LIN {X 0,Y 384.347,Z 411.583,A -85,B 0,C 180,E1 -11892.675,E2 -11892.675} C_VEL
LIN {X 0,Y 385.318,Z 404.439,A -85,B 0,C 180,E1 -11894.524,E2 -11894.524} C_VEL
LIN {X 0,Y 386.67,Z 395.805,A -85,B 0,C 180,E1 -11896.363,E2 -11896.363} C_VEL
LIN {X 0,Y 388.197,Z 385.439,A -85,B 0,C 180,E1 -11898.197,E2 -11898.197} C_VEL
LIN {X 0,Y 389.705,Z 374.807,A -85,B 0,C 180,E1 -11899.763,E2 -11899.763} C_VEL
LIN {X 0,Y 391.478,Z 362.137,A -85,B 0,C 180,E1 -11901.317,E2 -11901.317} C_VEL
LIN {X 0,Y 393.105,Z 349.489,A -85,B 0,C 180,E1 -11902.605,E2 -11902.605} C_VEL
LIN {X 0,Y 394.718,Z 335.76,A -85,B 0,C 180,E1 -11903.756,E2 -11903.756} C_VEL
LIN {X 0,Y 396.173,Z 321.35,A -85,B 0,C 180,E1 -11904.735,E2 -11904.735} C_VEL
LIN {X 0,Y 397.574,Z 305.833,A -85,B 0,C 180,E1 -11905.551,E2 -11905.551} C_VEL
LIN {X 0,Y 398.601,Z 290.565,A -85,B 0,C 180,E1 -11906.154,E2 -11906.154} C_VEL
LIN {X 0,Y 403.483,Z 217.535,A -85,B 0,C 180,E1 -11908.256,E2 -11908.256} C_VEL
LIN {X 0,Y 407.824,Z 166.369,A -85,B 0,C 180,E1 -11909.77,E2 -11909.77} C_VEL
LIN {X 0,Y 404.879,Z 160.3,A -85,B 0,C 180,E1 -11910.501,E2 -11910.501} C_VEL
LIN {X 0,Y 400.279,Z 152.554,A -85,B 0,C 180,E1 -11911.666,E2 -11911.666} C_VEL
LIN {X 0,Y 396.216,Z 146.476,A -85,B 0,C 180,E1 -11912.795,E2 -11912.795} C_VEL
LIN {X 0,Y 393.462,Z 142.689,A -85,B 0,C 180,E1 -11913.622,E2 -11913.622} C_VEL
LIN {X 0,Y 390.258,Z 138.514,A -85,B 0,C 180,E1 -11914.697,E2 -11914.697} C_VEL
LIN {X 0,Y 387.178,Z 134.685,A -85,B 0,C 180,E1 -11915.863,E2 -11915.863} C_VEL
LIN {X 0,Y 386.326,Z 132.28,A -85,B 0,C 180,E1 -11918.208,E2 -11918.208} C_VEL
LIN {X 0,Y 385.813,Z 130.877,A -85,B 0,C 180,E1 -11920.978,E2 -11920.978} C_VEL
LIN {X 0,Y 385.849,Z 130.902,A -85,B 0,C 180,E1 -11923.233,E2 -11923.233} C_VEL
LIN {X 0,Y 386.163,Z 131.856,A -85,B 0,C 180,E1 -11925.217,E2 -11925.217} C_VEL
LIN {X 0,Y 386.644,Z 133,A -85,B 0,C 180,E1 -11926.642,E2 -11926.642} C_VEL
LIN {X 0,Y 388.078,Z 136.761,A -85,B 0,C 180,E1 -11929.518,E2 -11929.518} C_VEL
LIN {X 0,Y 389.912,Z 141.995,A -85,B 0,C 180,E1 -11932.205,E2 -11932.205} C_VEL
LIN {X 0,Y 392.082,Z 149.259,A -85,B 0,C 180,E1 -11934.999,E2 -11934.999} C_VEL
LIN {X 0,Y 392.656,Z 151.099,A -85,B 0,C 180,E1 -11935.562,E2 -11935.562} C_VEL
LIN {X 0,Y 396.501,Z 158.649,A -85,B 0,C 180,E1 -11936.812,E2 -11936.812} C_VEL
LIN {X 0,Y 399.421,Z 164.695,A -85,B 0,C 180,E1 -11937.673,E2 -11937.673} C_VEL
LIN {X 0,Y 401.08,Z 168.627,A -85,B 0,C 180,E1 -11938.149,E2 -11938.149} C_VEL
LIN {X 0,Y 403.406,Z 182.486,A -85,B 0,C 180,E1 -11939.166,E2 -11939.166} C_VEL
LIN {X 0,Y 405.189,Z 197.13,A -85,B 0,C 180,E1 -11940.051,E2 -11940.051} C_VEL
LIN {X 0,Y 405.664,Z 204.273,A -85,B 0,C 180,E1 -11940.413,E2 -11940.413} C_VEL
LIN {X 0,Y 399.813,Z 285.015,A -85,B 0,C 180,E1 -11942.733,E2 -11942.733} C_VEL
LIN {X 0,Y 397.323,Z 326,A -85,B 0,C 180,E1 -11943.896,E2 -11943.896} C_VEL
LIN {X 0,Y 395.753,Z 342.836,A -85,B 0,C 180,E1 -11944.562,E2 -11944.562} C_VEL
LIN {X 0,Y 394.082,Z 357.859,A -85,B 0,C 180,E1 -11945.355,E2 -11945.355} C_VEL
LIN {X 0,Y 392.334,Z 372.724,A -85,B 0,C 180,E1 -11946.353,E2 -11946.353} C_VEL
LIN {X 0,Y 389.831,Z 393.298,A -85,B 0,C 180,E1 -11948.032,E2 -11948.032} C_VEL
LIN {X 0,Y 388.472,Z 405.12,A -85,B 0,C 180,E1 -11949.204,E2 -11949.204} C_VEL
LIN {X 0,Y 387.036,Z 417.181,A -85,B 0,C 180,E1 -11950.647,E2 -11950.647} C_VEL
LIN {X 0,Y 385.642,Z 428.175,A -85,B 0,C 180,E1 -11952.226,E2 -11952.226} C_VEL
LIN {X 0,Y 384.521,Z 437.485,A -85,B 0,C 180,E1 -11953.816,E2 -11953.816} C_VEL
LIN {X 0,Y 383.443,Z 446.573,A -85,B 0,C 180,E1 -11955.674,E2 -11955.674} C_VEL
LIN {X 0,Y 382.616,Z 455.061,A -85,B 0,C 180,E1 -11957.805,E2 -11957.805} C_VEL
LIN {X 0,Y 382.021,Z 461.857,A -85,B 0,C 180,E1 -11959.935,E2 -11959.935} C_VEL
LIN {X 0,Y 381.784,Z 467.162,A -85,B 0,C 180,E1 -11962.064,E2 -11962.064} C_VEL
LIN {X 0,Y 381.668,Z 470.632,A -85,B 0,C 180,E1 -11963.906,E2 -11963.906} C_VEL
LIN {X 0,Y 381.614,Z 473.177,A -85,B 0,C 180,E1 -11965.775,E2 -11965.775} C_VEL
LIN {X 0,Y 381.625,Z 474.929,A -85,B 0,C 180,E1 -11967.889,E2 -11967.889} C_VEL
LIN {X 0,Y 381.641,Z 475.494,A -85,B 0,C 180,E1 -11970,E2 -11970} C_VEL
LIN {X 0,Y 381.625,Z 474.855,A -85,B 0,C 180,E1 -11972.111,E2 -11972.111} C_VEL
LIN {X 0,Y 381.618,Z 472.984,A -85,B 0,C 180,E1 -11974.225,E2 -11974.225} C_VEL
LIN {X 0,Y 381.704,Z 469.874,A -85,B 0,C 180,E1 -11976.343,E2 -11976.343} C_VEL
LIN {X 0,Y 381.791,Z 465.448,A -85,B 0,C 180,E1 -11978.468,E2 -11978.468} C_VEL
LIN {X 0,Y 382.103,Z 459.605,A -85,B 0,C 180,E1 -11980.599,E2 -11980.599} C_VEL
LIN {X 0,Y 382.631,Z 453.192,A -85,B 0,C 180,E1 -11982.464,E2 -11982.464} C_VEL
LIN {X 0,Y 383.329,Z 445.398,A -85,B 0,C 180,E1 -11984.33,E2 -11984.33} C_VEL
LIN {X 0,Y 384.374,Z 435.976,A -85,B 0,C 180,E1 -11986.191,E2 -11986.191} C_VEL
LIN {X 0,Y 385.486,Z 426.338,A -85,B 0,C 180,E1 -11987.781,E2 -11987.781} C_VEL
LIN {X 0,Y 386.647,Z 415.895,A -85,B 0,C 180,E1 -11989.236,E2 -11989.236} C_VEL
LIN {X 0,Y 387.865,Z 404.637,A -85,B 0,C 180,E1 -11990.553,E2 -11990.553} C_VEL
LIN {X 0,Y 389.212,Z 392.493,A -85,B 0,C 180,E1 -11991.726,E2 -11991.726} C_VEL
LIN {X 0,Y 391.575,Z 372.289,A -85,B 0,C 180,E1 -11993.398,E2 -11993.398} C_VEL
LIN {X 0,Y 393.335,Z 357.326,A -85,B 0,C 180,E1 -11994.406,E2 -11994.406} C_VEL
LIN {X 0,Y 394.983,Z 341.955,A -85,B 0,C 180,E1 -11995.209,E2 -11995.209} C_VEL
LIN {X 0,Y 396.443,Z 325.504,A -85,B 0,C 180,E1 -11995.848,E2 -11995.848} C_VEL
LIN {X 0,Y 402.25,Z 235.432,A -85,B 0,C 180,E1 -11998.413,E2 -11998.413} C_VEL
LIN {X 0,Y 405.001,Z 198.369,A -85,B 0,C 180,E1 -11999.525,E2 -11999.525} C_VEL
LIN {X 0,Y 403.865,Z 178.688,A -85,B 0,C 180,E1 -12000.517,E2 -12000.517} C_VEL
LIN {X 0,Y 402.692,Z 165.49,A -85,B 0,C 180,E1 -12001.295,E2 -12001.295} C_VEL
LIN {X 0,Y 399.155,Z 154.868,A -85,B 0,C 180,E1 -12002.419,E2 -12002.419} C_VEL
LIN {X 0,Y 395.258,Z 143.156,A -85,B 0,C 180,E1 -12003.828,E2 -12003.828} C_VEL
LIN {X 0,Y 393.762,Z 140.224,A -85,B 0,C 180,E1 -12004.414,E2 -12004.414} C_VEL
LIN {X 0,Y 392.349,Z 137.801,A -85,B 0,C 180,E1 -12004.974,E2 -12004.974} C_VEL
LIN {X 0,Y 391.308,Z 136.6,A -85,B 0,C 180,E1 -12005.364,E2 -12005.364} C_VEL
LIN {X 0,Y 389.233,Z 133.196,A -85,B 0,C 180,E1 -12006.312,E2 -12006.312} C_VEL
LIN {X 0,Y 387.579,Z 131.177,A -85,B 0,C 180,E1 -12007.075,E2 -12007.075} C_VEL
LIN {X 0,Y 386.337,Z 128.589,A -85,B 0,C 180,E1 -12007.852,E2 -12007.852} C_VEL
LIN {X 0,Y 384.354,Z 126.735,A -85,B 0,C 180,E1 -12008.944,E2 -12008.944} C_VEL
LIN {X 0,Y 383.217,Z 124.543,A -85,B 0,C 180,E1 -12009.932,E2 -12009.932} C_VEL
LIN {X 0,Y 382.968,Z 123.404,A -85,B 0,C 180,E1 -12010.424,E2 -12010.424} C_VEL
LIN {X 0,Y 383.005,Z 123.401,A -85,B 0,C 180,E1 -12012.779,E2 -12012.779} C_VEL
LIN {X 0,Y 382.989,Z 123.398,A -85,B 0,C 180,E1 -12015.788,E2 -12015.788} C_VEL
LIN {X 0,Y 382.96,Z 123.404,A -85,B 0,C 180,E1 -12018.801,E2 -12018.801} C_VEL
LIN {X 0,Y 383.017,Z 123.514,A -85,B 0,C 180,E1 -12020.792,E2 -12020.792} C_VEL
LIN {X 0,Y 383.818,Z 125.952,A -85,B 0,C 180,E1 -12021.94,E2 -12021.94} C_VEL
LIN {X 0,Y 385.61,Z 128.057,A -85,B 0,C 180,E1 -12023.315,E2 -12023.315} C_VEL
LIN {X 0,Y 386.401,Z 130.05,A -85,B 0,C 180,E1 -12023.996,E2 -12023.996} C_VEL
LIN {X 0,Y 389.987,Z 134.512,A -85,B 0,C 180,E1 -12025.361,E2 -12025.361} C_VEL
LIN {X 0,Y 393.017,Z 138.694,A -85,B 0,C 180,E1 -12026.39,E2 -12026.39} C_VEL
LIN {X 0,Y 396.646,Z 144.079,A -85,B 0,C 180,E1 -12027.49,E2 -12027.49} C_VEL
LIN {X 0,Y 401.33,Z 151.497,A -85,B 0,C 180,E1 -12028.756,E2 -12028.756} C_VEL
LIN {X 0,Y 406.014,Z 160.362,A -85,B 0,C 180,E1 -12029.938,E2 -12029.938} C_VEL
LIN {X 0,Y 407.556,Z 163.653,A -85,B 0,C 180,E1 -12030.318,E2 -12030.318} C_VEL
LIN {X 0,Y 401.249,Z 243.859,A -85,B 0,C 180,E1 -12032.663,E2 -12032.663} C_VEL
LIN {X 0,Y 398.178,Z 293.464,A -85,B 0,C 180,E1 -12034.088,E2 -12034.088} C_VEL
LIN {X 0,Y 397.002,Z 309.399,A -85,B 0,C 180,E1 -12034.762,E2 -12034.762} C_VEL
LIN {X 0,Y 395.647,Z 324.606,A -85,B 0,C 180,E1 -12035.623,E2 -12035.623} C_VEL
LIN {X 0,Y 394.22,Z 338.624,A -85,B 0,C 180,E1 -12036.63,E2 -12036.63} C_VEL
LIN {X 0,Y 392.635,Z 351.845,A -85,B 0,C 180,E1 -12037.782,E2 -12037.782} C_VEL
LIN {X 0,Y 390.896,Z 365.316,A -85,B 0,C 180,E1 -12039.215,E2 -12039.215} C_VEL
LIN {X 0,Y 389.398,Z 375.479,A -85,B 0,C 180,E1 -12040.495,E2 -12040.495} C_VEL
LIN {X 0,Y 387.867,Z 385.981,A -85,B 0,C 180,E1 -12042.06,E2 -12042.06} C_VEL
LIN {X 0,Y 386.503,Z 396.196,A -85,B 0,C 180,E1 -12043.901,E2 -12043.901} C_VEL
LIN {X 0,Y 385.148,Z 404.718,A -85,B 0,C 180,E1 -12045.739,E2 -12045.739} C_VEL
LIN {X 0,Y 384.295,Z 410.874,A -85,B 0,C 180,E1 -12047.323,E2 -12047.323} C_VEL
LIN {X 0,Y 383.397,Z 417.548,A -85,B 0,C 180,E1 -12049.438,E2 -12049.438} C_VEL
LIN {X 0,Y 382.763,Z 422.72,A -85,B 0,C 180,E1 -12051.554,E2 -12051.554} C_VEL
LIN {X 0,Y 382.275,Z 426.502,A -85,B 0,C 180,E1 -12053.667,E2 -12053.667} C_VEL
LIN {X 0,Y 382.071,Z 428.972,A -85,B 0,C 180,E1 -12055.781,E2 -12055.781} C_VEL
LIN {X 0,Y 381.861,Z 430.199,A -85,B 0,C 180,E1 -12057.891,E2 -12057.891} C_VEL
LIN {X 0,Y 381.723,Z 430.189,A -85,B 0,C 180,E1 -12060,E2 -12060} C_VEL
LIN {X 0,Y 381.818,Z 428.931,A -85,B 0,C 180,E1 -12062.11,E2 -12062.11} C_VEL
LIN {X 0,Y 381.815,Z 426.423,A -85,B 0,C 180,E1 -12064.223,E2 -12064.223} C_VEL
LIN {X 0,Y 382.024,Z 422.597,A -85,B 0,C 180,E1 -12066.338,E2 -12066.338} C_VEL
LIN {X 0,Y 382.281,Z 417.372,A -85,B 0,C 180,E1 -12068.458,E2 -12068.458} C_VEL
LIN {X 0,Y 382.684,Z 410.604,A -85,B 0,C 180,E1 -12070.583,E2 -12070.583} C_VEL
LIN {X 0,Y 383.352,Z 403.259,A -85,B 0,C 180,E1 -12072.44,E2 -12072.44} C_VEL
LIN {X 0,Y 383.933,Z 394.641,A -85,B 0,C 180,E1 -12074.253,E2 -12074.253} C_VEL
LIN {X 0,Y 384.776,Z 385.298,A -85,B 0,C 180,E1 -12075.901,E2 -12075.901} C_VEL
LIN {X 0,Y 385.763,Z 374.58,A -85,B 0,C 180,E1 -12077.494,E2 -12077.494} C_VEL
LIN {X 0,Y 386.809,Z 362.92,A -85,B 0,C 180,E1 -12078.952,E2 -12078.952} C_VEL
LIN {X 0,Y 387.96,Z 350.303,A -85,B 0,C 180,E1 -12080.271,E2 -12080.271} C_VEL
LIN {X 0,Y 388.967,Z 336.567,A -85,B 0,C 180,E1 -12081.462,E2 -12081.462} C_VEL
LIN {X 0,Y 390.088,Z 321.475,A -85,B 0,C 180,E1 -12082.511,E2 -12082.511} C_VEL
LIN {X 0,Y 390.89,Z 307.073,A -85,B 0,C 180,E1 -12083.301,E2 -12083.301} C_VEL
LIN {X 0,Y 391.648,Z 290.801,A -85,B 0,C 180,E1 -12083.964,E2 -12083.964} C_VEL
LIN {X 0,Y 392.212,Z 273.108,A -85,B 0,C 180,E1 -12084.445,E2 -12084.445} C_VEL
LIN {X 0,Y 396.071,Z 155.461,A -85,B 0,C 180,E1 -12087.166,E2 -12087.166} C_VEL
LIN {X 0,Y 395.222,Z 152.536,A -85,B 0,C 180,E1 -12087.288,E2 -12087.288} C_VEL
LIN {X 0,Y 388.467,Z 136.45,A -85,B 0,C 180,E1 -12088.103,E2 -12088.103} C_VEL
LIN {X 0,Y 383.124,Z 124.081,A -85,B 0,C 180,E1 -12088.768,E2 -12088.768} C_VEL
LIN {X 0,Y 382.995,Z 123.402,A -85,B 0,C 180,E1 -12088.805,E2 -12088.805} C_VEL
LIN {X 0,Y 382.987,Z 123.403,A -85,B 0,C 180,E1 -12092.422,E2 -12092.422} C_VEL
LIN {X 0,Y 383.025,Z 123.399,A -85,B 0,C 180,E1 -12095.956,E2 -12095.956} C_VEL
LIN {X 0,Y 382.988,Z 123.405,A -85,B 0,C 180,E1 -12099.581,E2 -12099.581} C_VEL
LIN {X 0,Y 383.008,Z 123.4,A -85,B 0,C 180,E1 -12102.779,E2 -12102.779} C_VEL
LIN {X 0,Y 382.992,Z 123.38,A -85,B 0,C 180,E1 -12105.788,E2 -12105.788} C_VEL
LIN {X 0,Y 382.963,Z 123.397,A -85,B 0,C 180,E1 -12108.801,E2 -12108.801} C_VEL
LIN {X 0,Y 382.997,Z 123.397,A -85,B 0,C 180,E1 -12112.098,E2 -12112.098} C_VEL
LIN {X 0,Y 383.014,Z 123.387,A -85,B 0,C 180,E1 -12115.332,E2 -12115.332} C_VEL
LIN {X 0,Y 382.984,Z 123.397,A -85,B 0,C 180,E1 -12119.081,E2 -12119.081} C_VEL
LIN {X 0,Y 382.988,Z 123.402,A -85,B 0,C 180,E1 -12122.693,E2 -12122.693} C_VEL
LIN {X 0,Y 383.011,Z 123.388,A -85,B 0,C 180,E1 -12126.191,E2 -12126.191} C_VEL
LIN {X 0,Y 383.059,Z 123.388,A -85,B 0,C 180,E1 -12129.599,E2 -12129.599} C_VEL
LIN {X 0,Y 383.073,Z 123.389,A -85,B 0,C 180,E1 -12132.93,E2 -12132.93} C_VEL
LIN {X 0,Y 383.129,Z 123.383,A -85,B 0,C 180,E1 -12136.464,E2 -12136.464} C_VEL
LIN {X 0,Y 383.142,Z 123.386,A -85,B 0,C 180,E1 -12140.498,E2 -12140.498} C_VEL
LIN {X 0,Y 383.234,Z 123.372,A -85,B 0,C 180,E1 -12143.683,E2 -12143.683} C_VEL
LIN {X 0,Y 383.249,Z 123.435,A -85,B 0,C 180,E1 -12143.98,E2 -12143.98} C_VEL
LIN {X 0,Y 388.071,Z 141.249,A -85,B 0,C 180,E1 -12147.277,E2 -12147.277} C_VEL
LIN {X 0,Y 388.714,Z 143.994,A -85,B 0,C 180,E1 -12147.726,E2 -12147.726} C_VEL
LIN {X 0,Y 394.59,Z 158.144,A -85,B 0,C 180,E1 -12148.469,E2 -12148.469} C_VEL
LIN {X 0,Y 398.34,Z 176.527,A -85,B 0,C 180,E1 -12149.12,E2 -12149.12} C_VEL
LIN {X 0,Y 397.081,Z 229.861,A -85,B 0,C 180,E1 -12150.108,E2 -12150.108} C_VEL
LIN {X 0,Y 396.391,Z 235.707,A -85,B 0,C 180,E1 -12150.179,E2 -12150.179} C_VEL
LIN {X 0,Y 390.73,Z 254.736,A -85,B 0,C 180,E1 -12150.174,E2 -12150.174} C_VEL
LIN {X 0,Y 389.993,Z 260.586,A -85,B 0,C 180,E1 -12150.241,E2 -12150.241} C_VEL
LIN {X 0,Y 388.789,Z 311.527,A -85,B 0,C 180,E1 -12151.23,E2 -12151.23} C_VEL
LIN {X 0,Y 388.037,Z 326.659,A -85,B 0,C 180,E1 -12151.719,E2 -12151.719} C_VEL
LIN {X 0,Y 387.045,Z 341.921,A -85,B 0,C 180,E1 -12152.435,E2 -12152.435} C_VEL
LIN {X 0,Y 385.875,Z 355.419,A -85,B 0,C 180,E1 -12153.263,E2 -12153.263} C_VEL
LIN {X 0,Y 384.535,Z 369.093,A -85,B 0,C 180,E1 -12154.324,E2 -12154.324} C_VEL
LIN {X 0,Y 383.103,Z 381.72,A -85,B 0,C 180,E1 -12155.527,E2 -12155.527} C_VEL
LIN {X 0,Y 381.634,Z 393.46,A -85,B 0,C 180,E1 -12156.874,E2 -12156.874} C_VEL
LIN {X 0,Y 380.074,Z 405.246,A -85,B 0,C 180,E1 -12158.507,E2 -12158.507} C_VEL
LIN {X 0,Y 378.627,Z 416.121,A -85,B 0,C 180,E1 -12160.333,E2 -12160.333} C_VEL
LIN {X 0,Y 377.491,Z 424.838,A -85,B 0,C 180,E1 -12162.09,E2 -12162.09} C_VEL
LIN {X 0,Y 376.482,Z 432.891,A -85,B 0,C 180,E1 -12164.045,E2 -12164.045} C_VEL
LIN {X 0,Y 375.644,Z 440.368,A -85,B 0,C 180,E1 -12166.298,E2 -12166.298} C_VEL
LIN {X 0,Y 375.049,Z 446.256,A -85,B 0,C 180,E1 -12168.576,E2 -12168.576} C_VEL
LIN {X 0,Y 374.615,Z 450.693,A -85,B 0,C 180,E1 -12170.882,E2 -12170.882} C_VEL
LIN {X 0,Y 374.366,Z 453.731,A -85,B 0,C 180,E1 -12173.218,E2 -12173.218} C_VEL
LIN {X 0,Y 374.254,Z 455.426,A -85,B 0,C 180,E1 -12175.659,E2 -12175.659} C_VEL
LIN {X 0,Y 374.289,Z 455.655,A -85,B 0,C 180,E1 -12178.052,E2 -12178.052} C_VEL
LIN {X 0,Y 374.371,Z 454.465,A -85,B 0,C 180,E1 -12180.455,E2 -12180.455} C_VEL
LIN {X 0,Y 374.556,Z 452.434,A -85,B 0,C 180,E1 -12182.396,E2 -12182.396} C_VEL
LIN {X 0,Y 374.89,Z 449.297,A -85,B 0,C 180,E1 -12184.425,E2 -12184.425} C_VEL
LIN {X 0,Y 375.298,Z 445.262,A -85,B 0,C 180,E1 -12186.366,E2 -12186.366} C_VEL
LIN {X 0,Y 375.858,Z 440.242,A -85,B 0,C 180,E1 -12188.247,E2 -12188.247} C_VEL
LIN {X 0,Y 376.767,Z 433.239,A -85,B 0,C 180,E1 -12190.367,E2 -12190.367} C_VEL
LIN {X 0,Y 377.887,Z 424.993,A -85,B 0,C 180,E1 -12192.391,E2 -12192.391} C_VEL
LIN {X 0,Y 379.386,Z 414.89,A -85,B 0,C 180,E1 -12194.416,E2 -12194.416} C_VEL
LIN {X 0,Y 380.939,Z 404.013,A -85,B 0,C 180,E1 -12196.205,E2 -12196.205} C_VEL
LIN {X 0,Y 382.479,Z 393.101,A -85,B 0,C 180,E1 -12197.696,E2 -12197.696} C_VEL
LIN {X 0,Y 384.18,Z 380.61,A -85,B 0,C 180,E1 -12199.113,E2 -12199.113} C_VEL
LIN {X 0,Y 385.851,Z 366.742,A -85,B 0,C 180,E1 -12200.394,E2 -12200.394} C_VEL
LIN {X 0,Y 387.307,Z 352.562,A -85,B 0,C 180,E1 -12201.444,E2 -12201.444} C_VEL
LIN {X 0,Y 388.566,Z 338.284,A -85,B 0,C 180,E1 -12202.268,E2 -12202.268} C_VEL
LIN {X 0,Y 389.523,Z 323.755,A -85,B 0,C 180,E1 -12202.897,E2 -12202.897} C_VEL
LIN {X 0,Y 390.263,Z 308.063,A -85,B 0,C 180,E1 -12203.352,E2 -12203.352} C_VEL
LIN {X 0,Y 393.656,Z 171.803,A -85,B 0,C 180,E1 -12205.967,E2 -12205.967} C_VEL
LIN {X 0,Y 392.316,Z 164.643,A -85,B 0,C 180,E1 -12206.239,E2 -12206.239} C_VEL
LIN {X 0,Y 384.1,Z 146.331,A -85,B 0,C 180,E1 -12207.394,E2 -12207.394} C_VEL
LIN {X 0,Y 382.333,Z 142.759,A -85,B 0,C 180,E1 -12207.66,E2 -12207.66} C_VEL
LIN {X 0,Y 377.259,Z 127.998,A -85,B 0,C 180,E1 -12210.11,E2 -12210.11} C_VEL
LIN {X 0,Y 375.991,Z 124.27,A -85,B 0,C 180,E1 -12210.769,E2 -12210.769} C_VEL
LIN {X 0,Y 376.017,Z 124.514,A -85,B 0,C 180,E1 -12210.824,E2 -12210.824} C_VEL
LIN {X 0,Y 378.083,Z 129.65,A -85,B 0,C 180,E1 -12211.098,E2 -12211.098} C_VEL
LIN {X 0,Y 389.455,Z 155.72,A -85,B 0,C 180,E1 -12212.497,E2 -12212.497} C_VEL
LIN {X 0,Y 387.13,Z 223.764,A -85,B 0,C 180,E1 -12214.134,E2 -12214.134} C_VEL
LIN {X 0,Y 385.087,Z 287.202,A -85,B 0,C 180,E1 -12215.671,E2 -12215.671} C_VEL
LIN {X 0,Y 384.388,Z 303.256,A -85,B 0,C 180,E1 -12216.281,E2 -12216.281} C_VEL
LIN {X 0,Y 383.509,Z 318.597,A -85,B 0,C 180,E1 -12217.081,E2 -12217.081} C_VEL
LIN {X 0,Y 382.52,Z 332.61,A -85,B 0,C 180,E1 -12218.016,E2 -12218.016} C_VEL
LIN {X 0,Y 381.339,Z 347.144,A -85,B 0,C 180,E1 -12219.22,E2 -12219.22} C_VEL
LIN {X 0,Y 380.182,Z 360.401,A -85,B 0,C 180,E1 -12220.564,E2 -12220.564} C_VEL
LIN {X 0,Y 379.094,Z 372.562,A -85,B 0,C 180,E1 -12222.048,E2 -12222.048} C_VEL
LIN {X 0,Y 377.98,Z 384.555,A -85,B 0,C 180,E1 -12223.805,E2 -12223.805} C_VEL
LIN {X 0,Y 377.069,Z 394.12,A -85,B 0,C 180,E1 -12225.481,E2 -12225.481} C_VEL
LIN {X 0,Y 376.427,Z 402.939,A -85,B 0,C 180,E1 -12227.327,E2 -12227.327} C_VEL
LIN {X 0,Y 375.698,Z 410.47,A -85,B 0,C 180,E1 -12229.218,E2 -12229.218} C_VEL
LIN {X 0,Y 375.263,Z 417.429,A -85,B 0,C 180,E1 -12231.383,E2 -12231.383} C_VEL
LIN {X 0,Y 374.952,Z 422.824,A -85,B 0,C 180,E1 -12233.542,E2 -12233.542} C_VEL
LIN {X 0,Y 374.766,Z 426.803,A -85,B 0,C 180,E1 -12235.698,E2 -12235.698} C_VEL
LIN {X 0,Y 374.767,Z 429.461,A -85,B 0,C 180,E1 -12237.85,E2 -12237.85} C_VEL
LIN {X 0,Y 374.662,Z 430.875,A -85,B 0,C 180,E1 -12240,E2 -12240} C_VEL
LIN {X 0,Y 374.815,Z 431.039,A -85,B 0,C 180,E1 -12242.149,E2 -12242.149} C_VEL
LIN {X 0,Y 375.04,Z 429.938,A -85,B 0,C 180,E1 -12244.298,E2 -12244.298} C_VEL
LIN {X 0,Y 375.272,Z 427.593,A -85,B 0,C 180,E1 -12246.451,E2 -12246.451} C_VEL
LIN {X 0,Y 375.782,Z 423.956,A -85,B 0,C 180,E1 -12248.605,E2 -12248.605} C_VEL
LIN {X 0,Y 376.507,Z 418.961,A -85,B 0,C 180,E1 -12250.758,E2 -12250.758} C_VEL
LIN {X 0,Y 377.471,Z 412.493,A -85,B 0,C 180,E1 -12252.91,E2 -12252.91} C_VEL
LIN {X 0,Y 378.516,Z 405.458,A -85,B 0,C 180,E1 -12254.791,E2 -12254.791} C_VEL
LIN {X 0,Y 379.971,Z 396.957,A -85,B 0,C 180,E1 -12256.66,E2 -12256.66} C_VEL
LIN {X 0,Y 381.575,Z 386.751,A -85,B 0,C 180,E1 -12258.525,E2 -12258.525} C_VEL
LIN {X 0,Y 383.197,Z 376.3,A -85,B 0,C 180,E1 -12260.113,E2 -12260.113} C_VEL
LIN {X 0,Y 385.085,Z 363.87,A -85,B 0,C 180,E1 -12261.689,E2 -12261.689} C_VEL
LIN {X 0,Y 386.765,Z 351.534,A -85,B 0,C 180,E1 -12262.997,E2 -12262.997} C_VEL
LIN {X 0,Y 388.691,Z 336.604,A -85,B 0,C 180,E1 -12264.289,E2 -12264.289} C_VEL
LIN {X 0,Y 390.314,Z 321.779,A -85,B 0,C 180,E1 -12265.318,E2 -12265.318} C_VEL
LIN {X 0,Y 391.834,Z 306.159,A -85,B 0,C 180,E1 -12266.153,E2 -12266.153} C_VEL
LIN {X 0,Y 392.924,Z 290.783,A -85,B 0,C 180,E1 -12266.776,E2 -12266.776} C_VEL
LIN {X 0,Y 398.229,Z 218.568,A -85,B 0,C 180,E1 -12268.925,E2 -12268.925} C_VEL
LIN {X 0,Y 402.768,Z 169.117,A -85,B 0,C 180,E1 -12270.431,E2 -12270.431} C_VEL
LIN {X 0,Y 398.364,Z 160.786,A -85,B 0,C 180,E1 -12271.598,E2 -12271.598} C_VEL
LIN {X 0,Y 393.645,Z 153.189,A -85,B 0,C 180,E1 -12272.952,E2 -12272.952} C_VEL
LIN {X 0,Y 390.165,Z 148.367,A -85,B 0,C 180,E1 -12274.045,E2 -12274.045} C_VEL
LIN {X 0,Y 387.621,Z 144.861,A -85,B 0,C 180,E1 -12274.95,E2 -12274.95} C_VEL
LIN {X 0,Y 384.178,Z 140.696,A -85,B 0,C 180,E1 -12276.316,E2 -12276.316} C_VEL
LIN {X 0,Y 380.666,Z 136.62,A -85,B 0,C 180,E1 -12278.057,E2 -12278.057} C_VEL
LIN {X 0,Y 380.17,Z 135.256,A -85,B 0,C 180,E1 -12280.717,E2 -12280.717} C_VEL
LIN {X 0,Y 380.211,Z 135.183,A -85,B 0,C 180,E1 -12283.151,E2 -12283.151} C_VEL
LIN {X 0,Y 380.769,Z 136.795,A -85,B 0,C 180,E1 -12286.041,E2 -12286.041} C_VEL
LIN {X 0,Y 381.76,Z 139.538,A -85,B 0,C 180,E1 -12288.491,E2 -12288.491} C_VEL
LIN {X 0,Y 382.881,Z 142.588,A -85,B 0,C 180,E1 -12290.437,E2 -12290.437} C_VEL
LIN {X 0,Y 384.589,Z 147.783,A -85,B 0,C 180,E1 -12292.912,E2 -12292.912} C_VEL
LIN {X 0,Y 385.142,Z 149.526,A -85,B 0,C 180,E1 -12293.533,E2 -12293.533} C_VEL
LIN {X 0,Y 389.644,Z 157.429,A -85,B 0,C 180,E1 -12295.265,E2 -12295.265} C_VEL
LIN {X 0,Y 393.056,Z 164.36,A -85,B 0,C 180,E1 -12296.428,E2 -12296.428} C_VEL
LIN {X 0,Y 395.593,Z 169.872,A -85,B 0,C 180,E1 -12297.233,E2 -12297.233} C_VEL
LIN {X 0,Y 396.71,Z 172.826,A -85,B 0,C 180,E1 -12297.595,E2 -12297.595} C_VEL
LIN {X 0,Y 398.724,Z 186.14,A -85,B 0,C 180,E1 -12298.59,E2 -12298.59} C_VEL
LIN {X 0,Y 400.158,Z 199.615,A -85,B 0,C 180,E1 -12299.428,E2 -12299.428} C_VEL
LIN {X 0,Y 400.494,Z 205.625,A -85,B 0,C 180,E1 -12299.74,E2 -12299.74} C_VEL
LIN {X 0,Y 394.463,Z 281.862,A -85,B 0,C 180,E1 -12302.007,E2 -12302.007} C_VEL
LIN {X 0,Y 391.534,Z 325.853,A -85,B 0,C 180,E1 -12303.301,E2 -12303.301} C_VEL
LIN {X 0,Y 389.779,Z 342.991,A -85,B 0,C 180,E1 -12304,E2 -12304} C_VEL
LIN {X 0,Y 387.873,Z 359,A -85,B 0,C 180,E1 -12304.878,E2 -12304.878} C_VEL
LIN {X 0,Y 385.957,Z 373.911,A -85,B 0,C 180,E1 -12305.922,E2 -12305.922} C_VEL
LIN {X 0,Y 383.767,Z 389.113,A -85,B 0,C 180,E1 -12307.24,E2 -12307.24} C_VEL
LIN {X 0,Y 381.997,Z 403.976,A -85,B 0,C 180,E1 -12308.693,E2 -12308.693} C_VEL
LIN {X 0,Y 380.417,Z 416.193,A -85,B 0,C 180,E1 -12310.156,E2 -12310.156} C_VEL
LIN {X 0,Y 379.052,Z 426.454,A -85,B 0,C 180,E1 -12311.627,E2 -12311.627} C_VEL
LIN {X 0,Y 377.643,Z 437.412,A -85,B 0,C 180,E1 -12313.513,E2 -12313.513} C_VEL
LIN {X 0,Y 376.501,Z 446.47,A -85,B 0,C 180,E1 -12315.404,E2 -12315.404} C_VEL
LIN {X 0,Y 375.592,Z 454.935,A -85,B 0,C 180,E1 -12317.574,E2 -12317.574} C_VEL
LIN {X 0,Y 374.983,Z 461.719,A -85,B 0,C 180,E1 -12319.744,E2 -12319.744} C_VEL
LIN {X 0,Y 374.704,Z 467.012,A -85,B 0,C 180,E1 -12321.913,E2 -12321.913} C_VEL
LIN {X 0,Y 374.571,Z 470.74,A -85,B 0,C 180,E1 -12323.946,E2 -12323.946} C_VEL
LIN {X 0,Y 374.517,Z 473.01,A -85,B 0,C 180,E1 -12325.695,E2 -12325.695} C_VEL
LIN {X 0,Y 374.521,Z 474.752,A -85,B 0,C 180,E1 -12327.849,E2 -12327.849} C_VEL
LIN {X 0,Y 374.556,Z 475.305,A -85,B 0,C 180,E1 -12330,E2 -12330} C_VEL
LIN {X 0,Y 374.521,Z 474.658,A -85,B 0,C 180,E1 -12332.151,E2 -12332.151} C_VEL
LIN {X 0,Y 374.543,Z 472.776,A -85,B 0,C 180,E1 -12334.304,E2 -12334.304} C_VEL
LIN {X 0,Y 374.621,Z 469.65,A -85,B 0,C 180,E1 -12336.463,E2 -12336.463} C_VEL
LIN {X 0,Y 374.719,Z 465.209,A -85,B 0,C 180,E1 -12338.629,E2 -12338.629} C_VEL
LIN {X 0,Y 375.074,Z 459.349,A -85,B 0,C 180,E1 -12340.8,E2 -12340.8} C_VEL
LIN {X 0,Y 375.643,Z 452.918,A -85,B 0,C 180,E1 -12342.699,E2 -12342.699} C_VEL
LIN {X 0,Y 376.382,Z 445.102,A -85,B 0,C 180,E1 -12344.601,E2 -12344.601} C_VEL
LIN {X 0,Y 377.485,Z 435.657,A -85,B 0,C 180,E1 -12346.495,E2 -12346.495} C_VEL
LIN {X 0,Y 378.635,Z 425.99,A -85,B 0,C 180,E1 -12348.114,E2 -12348.114} C_VEL
LIN {X 0,Y 379.895,Z 414.436,A -85,B 0,C 180,E1 -12349.732,E2 -12349.732} C_VEL
LIN {X 0,Y 381.355,Z 402.96,A -85,B 0,C 180,E1 -12351.061,E2 -12351.061} C_VEL
LIN {X 0,Y 383.932,Z 382.986,A -85,B 0,C 180,E1 -12353.034,E2 -12353.034} C_VEL
LIN {X 0,Y 385.721,Z 369.941,A -85,B 0,C 180,E1 -12354.093,E2 -12354.093} C_VEL
LIN {X 0,Y 387.499,Z 355.104,A -85,B 0,C 180,E1 -12355.084,E2 -12355.084} C_VEL
LIN {X 0,Y 389.279,Z 339.576,A -85,B 0,C 180,E1 -12355.892,E2 -12355.892} C_VEL
LIN {X 0,Y 390.834,Z 322.816,A -85,B 0,C 180,E1 -12356.535,E2 -12356.535} C_VEL
LIN {X 0,Y 396.578,Z 240.263,A -85,B 0,C 180,E1 -12358.947,E2 -12358.947} C_VEL
LIN {X 0,Y 399.858,Z 199.935,A -85,B 0,C 180,E1 -12360.187,E2 -12360.187} C_VEL
LIN {X 0,Y 398.918,Z 179.629,A -85,B 0,C 180,E1 -12361.25,E2 -12361.25} C_VEL
LIN {X 0,Y 398.044,Z 168.745,A -85,B 0,C 180,E1 -12361.93,E2 -12361.93} C_VEL
LIN {X 0,Y 395.104,Z 159.366,A -85,B 0,C 180,E1 -12362.953,E2 -12362.953} C_VEL
LIN {X 0,Y 391.245,Z 147.411,A -85,B 0,C 180,E1 -12364.462,E2 -12364.462} C_VEL
LIN {X 0,Y 388.485,Z 143.243,A -85,B 0,C 180,E1 -12365.412,E2 -12365.412} C_VEL
LIN {X 0,Y 385.525,Z 138.903,A -85,B 0,C 180,E1 -12366.669,E2 -12366.669} C_VEL
LIN {X 0,Y 383.2,Z 135.097,A -85,B 0,C 180,E1 -12367.942,E2 -12367.942} C_VEL
LIN {X 0,Y 381.018,Z 132.729,A -85,B 0,C 180,E1 -12369.222,E2 -12369.222} C_VEL
LIN {X 0,Y 379.595,Z 129.63,A -85,B 0,C 180,E1 -12370.616,E2 -12370.616} C_VEL
LIN {X 0,Y 378.031,Z 128.49,A -85,B 0,C 180,E1 -12372.012,E2 -12372.012} C_VEL
LIN {X 0,Y 377.055,Z 127.319,A -85,B 0,C 180,E1 -12373.603,E2 -12373.603} C_VEL
LIN {X 0,Y 376.714,Z 126.732,A -85,B 0,C 180,E1 -12375.148,E2 -12375.148} C_VEL
LIN {X 0,Y 376.773,Z 126.853,A -85,B 0,C 180,E1 -12376.675,E2 -12376.675} C_VEL
LIN {X 0,Y 377.205,Z 127.581,A -85,B 0,C 180,E1 -12378.182,E2 -12378.182} C_VEL
LIN {X 0,Y 378.116,Z 128.595,A -85,B 0,C 180,E1 -12379.646,E2 -12379.646} C_VEL
LIN {X 0,Y 379.287,Z 130.311,A -85,B 0,C 180,E1 -12381.1,E2 -12381.1} C_VEL
LIN {X 0,Y 379.919,Z 131.75,A -85,B 0,C 180,E1 -12381.77,E2 -12381.77} C_VEL
LIN {X 0,Y 382.865,Z 134.829,A -85,B 0,C 180,E1 -12383.253,E2 -12383.253} C_VEL
LIN {X 0,Y 386.158,Z 139.23,A -85,B 0,C 180,E1 -12384.664,E2 -12384.664} C_VEL
LIN {X 0,Y 389.989,Z 144.715,A -85,B 0,C 180,E1 -12386.057,E2 -12386.057} C_VEL
LIN {X 0,Y 394.14,Z 151.044,A -85,B 0,C 180,E1 -12387.366,E2 -12387.366} C_VEL
LIN {X 0,Y 397.982,Z 157.576,A -85,B 0,C 180,E1 -12388.462,E2 -12388.462} C_VEL
LIN {X 0,Y 401.985,Z 165.52,A -85,B 0,C 180,E1 -12389.535,E2 -12389.535} C_VEL
LIN {X 0,Y 402.499,Z 166.68,A -85,B 0,C 180,E1 -12389.672,E2 -12389.672} C_VEL
LIN {X 0,Y 395.761,Z 245.276,A -85,B 0,C 180,E1 -12392.036,E2 -12392.036} C_VEL
LIN {X 0,Y 392.469,Z 293.932,A -85,B 0,C 180,E1 -12393.485,E2 -12393.485} C_VEL
LIN {X 0,Y 391.216,Z 309.791,A -85,B 0,C 180,E1 -12394.168,E2 -12394.168} C_VEL
LIN {X 0,Y 389.705,Z 325.333,A -85,B 0,C 180,E1 -12395.068,E2 -12395.068} C_VEL
LIN {X 0,Y 388.163,Z 339.396,A -85,B 0,C 180,E1 -12396.102,E2 -12396.102} C_VEL
LIN {X 0,Y 386.292,Z 353.808,A -85,B 0,C 180,E1 -12397.398,E2 -12397.398} C_VEL
LIN {X 0,Y 384.384,Z 367.303,A -85,B 0,C 180,E1 -12398.886,E2 -12398.886} C_VEL
LIN {X 0,Y 382.586,Z 378.796,A -85,B 0,C 180,E1 -12400.413,E2 -12400.413} C_VEL
LIN {X 0,Y 381.049,Z 388.81,A -85,B 0,C 180,E1 -12402.005,E2 -12402.005} C_VEL
LIN {X 0,Y 379.526,Z 398.643,A -85,B 0,C 180,E1 -12403.873,E2 -12403.873} C_VEL
LIN {X 0,Y 378.15,Z 406.806,A -85,B 0,C 180,E1 -12405.744,E2 -12405.744} C_VEL
LIN {X 0,Y 377.192,Z 413.533,A -85,B 0,C 180,E1 -12407.627,E2 -12407.627} C_VEL
LIN {X 0,Y 376.329,Z 419.722,A -85,B 0,C 180,E1 -12409.781,E2 -12409.781} C_VEL
LIN {X 0,Y 375.637,Z 424.444,A -85,B 0,C 180,E1 -12411.934,E2 -12411.934} C_VEL
LIN {X 0,Y 375.247,Z 427.127,A -85,B 0,C 180,E1 -12413.548,E2 -12413.548} C_VEL
LIN {X 0,Y 375.006,Z 429.532,A -85,B 0,C 180,E1 -12415.701,E2 -12415.701} C_VEL
LIN {X 0,Y 374.799,Z 430.678,A -85,B 0,C 180,E1 -12417.851,E2 -12417.851} C_VEL
LIN {X 0,Y 374.652,Z 430.582,A -85,B 0,C 180,E1 -12420,E2 -12420} C_VEL
LIN {X 0,Y 374.735,Z 429.235,A -85,B 0,C 180,E1 -12422.15,E2 -12422.15} C_VEL
LIN {X 0,Y 374.739,Z 426.633,A -85,B 0,C 180,E1 -12424.303,E2 -12424.303} C_VEL
LIN {X 0,Y 374.995,Z 422.331,A -85,B 0,C 180,E1 -12426.633,E2 -12426.633} C_VEL
LIN {X 0,Y 375.217,Z 417.367,A -85,B 0,C 180,E1 -12428.618,E2 -12428.618} C_VEL
LIN {X 0,Y 375.643,Z 410.475,A -85,B 0,C 180,E1 -12430.784,E2 -12430.784} C_VEL
LIN {X 0,Y 376.35,Z 402.996,A -85,B 0,C 180,E1 -12432.675,E2 -12432.675} C_VEL
LIN {X 0,Y 377.021,Z 393.946,A -85,B 0,C 180,E1 -12434.576,E2 -12434.576} C_VEL
LIN {X 0,Y 377.859,Z 384.711,A -85,B 0,C 180,E1 -12436.2,E2 -12436.2} C_VEL
LIN {X 0,Y 378.904,Z 373.796,A -85,B 0,C 180,E1 -12437.821,E2 -12437.821} C_VEL
LIN {X 0,Y 379.922,Z 362.529,A -85,B 0,C 180,E1 -12439.235,E2 -12439.235} C_VEL
LIN {X 0,Y 381.179,Z 349.004,A -85,B 0,C 180,E1 -12440.648,E2 -12440.648} C_VEL
LIN {X 0,Y 382.251,Z 334.916,A -85,B 0,C 180,E1 -12441.859,E2 -12441.859} C_VEL
LIN {X 0,Y 383.357,Z 320.429,A -85,B 0,C 180,E1 -12442.857,E2 -12442.857} C_VEL
LIN {X 0,Y 384.162,Z 305.654,A -85,B 0,C 180,E1 -12443.662,E2 -12443.662} C_VEL
LIN {X 0,Y 384.859,Z 290.482,A -85,B 0,C 180,E1 -12444.278,E2 -12444.278} C_VEL
LIN {X 0,Y 385.462,Z 272.957,A -85,B 0,C 180,E1 -12444.759,E2 -12444.759} C_VEL
LIN {X 0,Y 389.376,Z 156.282,A -85,B 0,C 180,E1 -12447.53,E2 -12447.53} C_VEL
LIN {X 0,Y 383.471,Z 142.046,A -85,B 0,C 180,E1 -12448.263,E2 -12448.263} C_VEL
LIN {X 0,Y 376.052,Z 124.759,A -85,B 0,C 180,E1 -12449.196,E2 -12449.196} C_VEL
LIN {X 0,Y 375.958,Z 124.281,A -85,B 0,C 180,E1 -12449.234,E2 -12449.234} C_VEL
LIN {X 0,Y 375.95,Z 124.28,A -85,B 0,C 180,E1 -12452.829,E2 -12452.829} C_VEL
LIN {X 0,Y 375.958,Z 124.281,A -85,B 0,C 180,E1 -12455.416,E2 -12455.416} C_VEL
LIN {X 0,Y 375.937,Z 124.28,A -85,B 0,C 180,E1 -12458.263,E2 -12458.263} C_VEL
LIN {X 0,Y 375.919,Z 124.286,A -85,B 0,C 180,E1 -12461.598,E2 -12461.598} C_VEL
LIN {X 0,Y 375.923,Z 124.275,A -85,B 0,C 180,E1 -12464.731,E2 -12464.731} C_VEL
LIN {X 0,Y 375.918,Z 124.265,A -85,B 0,C 180,E1 -12467.698,E2 -12467.698} C_VEL
LIN {X 0,Y 375.938,Z 124.28,A -85,B 0,C 180,E1 -12470.534,E2 -12470.534} C_VEL
LIN {X 0,Y 375.961,Z 124.26,A -85,B 0,C 180,E1 -12473.497,E2 -12473.497} C_VEL
LIN {X 0,Y 375.96,Z 124.272,A -85,B 0,C 180,E1 -12475.888,E2 -12475.888} C_VEL
LIN {X 0,Y 375.964,Z 124.267,A -85,B 0,C 180,E1 -12479.687,E2 -12479.687} C_VEL
LIN {X 0,Y 375.93,Z 124.277,A -85,B 0,C 180,E1 -12482.136,E2 -12482.136} C_VEL
LIN {X 0,Y 375.939,Z 124.279,A -85,B 0,C 180,E1 -12484.534,E2 -12484.534} C_VEL
LIN {X 0,Y 375.974,Z 124.271,A -85,B 0,C 180,E1 -12486.887,E2 -12486.887} C_VEL
LIN {X 0,Y 375.989,Z 124.267,A -85,B 0,C 180,E1 -12490.339,E2 -12490.339} C_VEL
LIN {X 0,Y 375.977,Z 124.269,A -85,B 0,C 180,E1 -12493.717,E2 -12493.717} C_VEL
LIN {X 0,Y 376.107,Z 124.256,A -85,B 0,C 180,E1 -12497.042,E2 -12497.042} C_VEL
LIN {X 0,Y 376.113,Z 124.259,A -85,B 0,C 180,E1 -12500.318,E2 -12500.318} C_VEL
LIN {X 0,Y 376.202,Z 124.377,A -85,B 0,C 180,E1 -12503.497,E2 -12503.497} C_VEL
LIN {X 0,Y 381.506,Z 143.772,A -85,B 0,C 180,E1 -12507.146,E2 -12507.146} C_VEL
LIN {X 0,Y 388.629,Z 161.191,A -85,B 0,C 180,E1 -12508.083,E2 -12508.083} C_VEL
LIN {X 0,Y 391.897,Z 176.955,A -85,B 0,C 180,E1 -12508.659,E2 -12508.659} C_VEL
LIN {X 0,Y 389.993,Z 260.586,A -85,B 0,C 180,E1 -12510.241,E2 -12510.241} C_VEL
LIN {X 0,Y 389.258,Z 266.434,A -85,B 0,C 180,E1 -12510.309,E2 -12510.309} C_VEL
LIN {X 0,Y 383.573,Z 285.456,A -85,B 0,C 180,E1 -12510.304,E2 -12510.304} C_VEL
LIN {X 0,Y 382.853,Z 291.303,A -85,B 0,C 180,E1 -12510.375,E2 -12510.375} C_VEL
LIN {X 0,Y 382.275,Z 312.615,A -85,B 0,C 180,E1 -12510.823,E2 -12510.823} C_VEL
LIN {X 0,Y 381.467,Z 328.219,A -85,B 0,C 180,E1 -12511.353,E2 -12511.353} C_VEL
LIN {X 0,Y 380.374,Z 343.821,A -85,B 0,C 180,E1 -12512.118,E2 -12512.118} C_VEL
LIN {X 0,Y 379.19,Z 356.875,A -85,B 0,C 180,E1 -12512.955,E2 -12512.955} C_VEL
LIN {X 0,Y 377.833,Z 369.943,A -85,B 0,C 180,E1 -12514,E2 -12514} C_VEL
LIN {X 0,Y 376.36,Z 382.453,A -85,B 0,C 180,E1 -12515.223,E2 -12515.223} C_VEL
LIN {X 0,Y 374.718,Z 394.952,A -85,B 0,C 180,E1 -12516.704,E2 -12516.704} C_VEL
LIN {X 0,Y 373.08,Z 406.721,A -85,B 0,C 180,E1 -12518.395,E2 -12518.395} C_VEL
LIN {X 0,Y 371.627,Z 417.144,A -85,B 0,C 180,E1 -12520.206,E2 -12520.206} C_VEL
LIN {X 0,Y 370.432,Z 425.946,A -85,B 0,C 180,E1 -12522.046,E2 -12522.046} C_VEL
LIN {X 0,Y 369.421,Z 433.744,A -85,B 0,C 180,E1 -12524.011,E2 -12524.011} C_VEL
LIN {X 0,Y 368.643,Z 440.353,A -85,B 0,C 180,E1 -12526.048,E2 -12526.048} C_VEL
LIN {X 0,Y 368.01,Z 446.285,A -85,B 0,C 180,E1 -12528.367,E2 -12528.367} C_VEL
LIN {X 0,Y 367.602,Z 450.381,A -85,B 0,C 180,E1 -12530.476,E2 -12530.476} C_VEL
LIN {X 0,Y 367.332,Z 453.24,A -85,B 0,C 180,E1 -12532.498,E2 -12532.498} C_VEL
LIN {X 0,Y 367.167,Z 455.286,A -85,B 0,C 180,E1 -12534.904,E2 -12534.904} C_VEL
LIN {X 0,Y 367.144,Z 455.94,A -85,B 0,C 180,E1 -12537.35,E2 -12537.35} C_VEL
LIN {X 0,Y 367.194,Z 455.728,A -85,B 0,C 180,E1 -12538.587,E2 -12538.587} C_VEL
LIN {X 0,Y 367.278,Z 454.641,A -85,B 0,C 180,E1 -12540.56,E2 -12540.56} C_VEL
LIN {X 0,Y 367.515,Z 452.383,A -85,B 0,C 180,E1 -12542.709,E2 -12542.709} C_VEL
LIN {X 0,Y 367.932,Z 448.791,A -85,B 0,C 180,E1 -12544.963,E2 -12544.963} C_VEL
LIN {X 0,Y 368.429,Z 444.087,A -85,B 0,C 180,E1 -12547.123,E2 -12547.123} C_VEL
LIN {X 0,Y 369.175,Z 438.064,A -85,B 0,C 180,E1 -12549.271,E2 -12549.271} C_VEL
LIN {X 0,Y 370.155,Z 430.898,A -85,B 0,C 180,E1 -12551.324,E2 -12551.324} C_VEL
LIN {X 0,Y 371.46,Z 422.448,A -85,B 0,C 180,E1 -12553.302,E2 -12553.302} C_VEL
LIN {X 0,Y 372.825,Z 413.855,A -85,B 0,C 180,E1 -12554.983,E2 -12554.983} C_VEL
LIN {X 0,Y 374.382,Z 403.369,A -85,B 0,C 180,E1 -12556.705,E2 -12556.705} C_VEL
LIN {X 0,Y 375.895,Z 393.118,A -85,B 0,C 180,E1 -12558.123,E2 -12558.123} C_VEL
LIN {X 0,Y 377.667,Z 380.493,A -85,B 0,C 180,E1 -12559.574,E2 -12559.574} C_VEL
LIN {X 0,Y 379.396,Z 366.76,A -85,B 0,C 180,E1 -12560.858,E2 -12560.858} C_VEL
LIN {X 0,Y 380.853,Z 353.408,A -85,B 0,C 180,E1 -12561.866,E2 -12561.866} C_VEL
LIN {X 0,Y 382.187,Z 339.184,A -85,B 0,C 180,E1 -12562.708,E2 -12562.708} C_VEL
LIN {X 0,Y 383.231,Z 324.16,A -85,B 0,C 180,E1 -12563.372,E2 -12563.372} C_VEL
LIN {X 0,Y 383.986,Z 308.545,A -85,B 0,C 180,E1 -12563.836,E2 -12563.836} C_VEL
LIN {X 0,Y 387.579,Z 173.195,A -85,B 0,C 180,E1 -12566.472,E2 -12566.472} C_VEL
LIN {X 0,Y 386.555,Z 167.556,A -85,B 0,C 180,E1 -12566.69,E2 -12566.69} C_VEL
LIN {X 0,Y 378.877,Z 150.258,A -85,B 0,C 180,E1 -12567.808,E2 -12567.808} C_VEL
LIN {X 0,Y 375.172,Z 142.888,A -85,B 0,C 180,E1 -12568.364,E2 -12568.364} C_VEL
LIN {X 0,Y 370.587,Z 129.983,A -85,B 0,C 180,E1 -12570.561,E2 -12570.561} C_VEL
LIN {X 0,Y 370.639,Z 129.91,A -85,B 0,C 180,E1 -12570.623,E2 -12570.623} C_VEL
LIN {X 0,Y 382.863,Z 157.524,A -85,B 0,C 180,E1 -12572.152,E2 -12572.152} C_VEL
LIN {X 0,Y 378.328,Z 286.905,A -85,B 0,C 180,E1 -12575.352,E2 -12575.352} C_VEL
LIN {X 0,Y 377.569,Z 303.117,A -85,B 0,C 180,E1 -12575.972,E2 -12575.972} C_VEL
LIN {X 0,Y 376.696,Z 318.559,A -85,B 0,C 180,E1 -12576.788,E2 -12576.788} C_VEL
LIN {X 0,Y 375.668,Z 332.641,A -85,B 0,C 180,E1 -12577.738,E2 -12577.738} C_VEL
LIN {X 0,Y 374.456,Z 347.238,A -85,B 0,C 180,E1 -12578.964,E2 -12578.964} C_VEL
LIN {X 0,Y 373.272,Z 360.173,A -85,B 0,C 180,E1 -12580.289,E2 -12580.289} C_VEL
LIN {X 0,Y 372.13,Z 372.755,A -85,B 0,C 180,E1 -12581.843,E2 -12581.843} C_VEL
LIN {X 0,Y 371.075,Z 383.942,A -85,B 0,C 180,E1 -12583.495,E2 -12583.495} C_VEL
LIN {X 0,Y 370.006,Z 394.825,A -85,B 0,C 180,E1 -12585.423,E2 -12585.423} C_VEL
LIN {X 0,Y 369.327,Z 403.843,A -85,B 0,C 180,E1 -12587.359,E2 -12587.359} C_VEL
LIN {X 0,Y 368.658,Z 410.329,A -85,B 0,C 180,E1 -12589.01,E2 -12589.01} C_VEL
LIN {X 0,Y 368.205,Z 417.414,A -85,B 0,C 180,E1 -12591.216,E2 -12591.216} C_VEL
LIN {X 0,Y 367.881,Z 422.925,A -85,B 0,C 180,E1 -12593.418,E2 -12593.418} C_VEL
LIN {X 0,Y 367.691,Z 427.01,A -85,B 0,C 180,E1 -12595.615,E2 -12595.615} C_VEL
LIN {X 0,Y 367.686,Z 429.772,A -85,B 0,C 180,E1 -12597.809,E2 -12597.809} C_VEL
LIN {X 0,Y 367.593,Z 431.28,A -85,B 0,C 180,E1 -12600,E2 -12600} C_VEL
LIN {X 0,Y 367.755,Z 431.511,A -85,B 0,C 180,E1 -12602.19,E2 -12602.19} C_VEL
LIN {X 0,Y 367.977,Z 430.489,A -85,B 0,C 180,E1 -12604.381,E2 -12604.381} C_VEL
LIN {X 0,Y 368.249,Z 428.239,A -85,B 0,C 180,E1 -12606.575,E2 -12606.575} C_VEL
LIN {X 0,Y 368.811,Z 424.692,A -85,B 0,C 180,E1 -12608.768,E2 -12608.768} C_VEL
LIN {X 0,Y 369.556,Z 419.808,A -85,B 0,C 180,E1 -12610.963,E2 -12610.963} C_VEL
LIN {X 0,Y 370.603,Z 413.449,A -85,B 0,C 180,E1 -12613.153,E2 -12613.153} C_VEL
LIN {X 0,Y 371.73,Z 406.539,A -85,B 0,C 180,E1 -12615.067,E2 -12615.067} C_VEL
LIN {X 0,Y 373.288,Z 398.182,A -85,B 0,C 180,E1 -12616.967,E2 -12616.967} C_VEL
LIN {X 0,Y 374.982,Z 388.149,A -85,B 0,C 180,E1 -12618.863,E2 -12618.863} C_VEL
LIN {X 0,Y 376.707,Z 377.902,A -85,B 0,C 180,E1 -12620.475,E2 -12620.475} C_VEL
LIN {X 0,Y 378.723,Z 365.73,A -85,B 0,C 180,E1 -12622.072,E2 -12622.072} C_VEL
LIN {X 0,Y 380.682,Z 352.403,A -85,B 0,C 180,E1 -12623.53,E2 -12623.53} C_VEL
LIN {X 0,Y 382.733,Z 337.659,A -85,B 0,C 180,E1 -12624.837,E2 -12624.837} C_VEL
LIN {X 0,Y 384.572,Z 322.112,A -85,B 0,C 180,E1 -12625.941,E2 -12625.941} C_VEL
LIN {X 0,Y 386.248,Z 305.868,A -85,B 0,C 180,E1 -12626.819,E2 -12626.819} C_VEL
LIN {X 0,Y 387.422,Z 290.652,A -85,B 0,C 180,E1 -12627.444,E2 -12627.444} C_VEL
LIN {X 0,Y 393.26,Z 218.523,A -85,B 0,C 180,E1 -12629.657,E2 -12629.657} C_VEL
LIN {X 0,Y 397.736,Z 172.094,A -85,B 0,C 180,E1 -12631.135,E2 -12631.135} C_VEL
LIN {X 0,Y 393.764,Z 164.554,A -85,B 0,C 180,E1 -12632.28,E2 -12632.28} C_VEL
LIN {X 0,Y 389.679,Z 158.042,A -85,B 0,C 180,E1 -12633.538,E2 -12633.538} C_VEL
LIN {X 0,Y 386.995,Z 154.121,A -85,B 0,C 180,E1 -12634.456,E2 -12634.456} C_VEL
LIN {X 0,Y 384.867,Z 151.129,A -85,B 0,C 180,E1 -12635.252,E2 -12635.252} C_VEL
LIN {X 0,Y 381.443,Z 146.924,A -85,B 0,C 180,E1 -12636.693,E2 -12636.693} C_VEL
LIN {X 0,Y 378.182,Z 143.108,A -85,B 0,C 180,E1 -12638.403,E2 -12638.403} C_VEL
LIN {X 0,Y 374.856,Z 139.918,A -85,B 0,C 180,E1 -12640.855,E2 -12640.855} C_VEL
LIN {X 0,Y 374.499,Z 139.406,A -85,B 0,C 180,E1 -12641.353,E2 -12641.353} C_VEL
LIN {X 0,Y 374.651,Z 139.797,A -85,B 0,C 180,E1 -12643.953,E2 -12643.953} C_VEL
LIN {X 0,Y 375.157,Z 141.181,A -85,B 0,C 180,E1 -12646.121,E2 -12646.121} C_VEL
LIN {X 0,Y 376.032,Z 143.655,A -85,B 0,C 180,E1 -12648.382,E2 -12648.382} C_VEL
LIN {X 0,Y 377.265,Z 146.984,A -85,B 0,C 180,E1 -12650.456,E2 -12650.456} C_VEL
LIN {X 0,Y 382.051,Z 154.985,A -85,B 0,C 180,E1 -12653.037,E2 -12653.037} C_VEL
LIN {X 0,Y 386.412,Z 163.161,A -85,B 0,C 180,E1 -12654.855,E2 -12654.855} C_VEL
LIN {X 0,Y 389.577,Z 169.932,A -85,B 0,C 180,E1 -12656.021,E2 -12656.021} C_VEL
LIN {X 0,Y 392.093,Z 175.707,A -85,B 0,C 180,E1 -12656.873,E2 -12656.873} C_VEL
LIN {X 0,Y 392.809,Z 179.153,A -85,B 0,C 180,E1 -12657.195,E2 -12657.195} C_VEL
LIN {X 0,Y 394.613,Z 193.833,A -85,B 0,C 180,E1 -12658.27,E2 -12658.27} C_VEL
LIN {X 0,Y 395.515,Z 206.467,A -85,B 0,C 180,E1 -12659.021,E2 -12659.021} C_VEL
LIN {X 0,Y 388.997,Z 282.512,A -85,B 0,C 180,E1 -12661.358,E2 -12661.358} C_VEL
LIN {X 0,Y 385.871,Z 325.349,A -85,B 0,C 180,E1 -12662.657,E2 -12662.657} C_VEL
LIN {X 0,Y 384.023,Z 342.188,A -85,B 0,C 180,E1 -12663.361,E2 -12663.361} C_VEL
LIN {X 0,Y 381.989,Z 358.003,A -85,B 0,C 180,E1 -12664.237,E2 -12664.237} C_VEL
LIN {X 0,Y 379.813,Z 373.921,A -85,B 0,C 180,E1 -12665.374,E2 -12665.374} C_VEL
LIN {X 0,Y 377.516,Z 388.796,A -85,B 0,C 180,E1 -12666.697,E2 -12666.697} C_VEL
LIN {X 0,Y 374.71,Z 408.682,A -85,B 0,C 180,E1 -12668.835,E2 -12668.835} C_VEL
LIN {X 0,Y 373.146,Z 420.191,A -85,B 0,C 180,E1 -12670.342,E2 -12670.342} C_VEL
LIN {X 0,Y 371.573,Z 431.355,A -85,B 0,C 180,E1 -12672.1,E2 -12672.1} C_VEL
LIN {X 0,Y 370.224,Z 441.426,A -85,B 0,C 180,E1 -12674.023,E2 -12674.023} C_VEL
LIN {X 0,Y 369.109,Z 450.266,A -85,B 0,C 180,E1 -12676.078,E2 -12676.078} C_VEL
LIN {X 0,Y 368.453,Z 456.652,A -85,B 0,C 180,E1 -12677.888,E2 -12677.888} C_VEL
LIN {X 0,Y 367.842,Z 463.028,A -85,B 0,C 180,E1 -12680.099,E2 -12680.099} C_VEL
LIN {X 0,Y 367.572,Z 467.944,A -85,B 0,C 180,E1 -12682.308,E2 -12682.308} C_VEL
LIN {X 0,Y 367.439,Z 471.525,A -85,B 0,C 180,E1 -12684.512,E2 -12684.512} C_VEL
LIN {X 0,Y 367.389,Z 473.858,A -85,B 0,C 180,E1 -12686.71,E2 -12686.71} C_VEL
LIN {X 0,Y 367.431,Z 474.993,A -85,B 0,C 180,E1 -12688.904,E2 -12688.904} C_VEL
LIN {X 0,Y 367.431,Z 474.939,A -85,B 0,C 180,E1 -12691.096,E2 -12691.096} C_VEL
LIN {X 0,Y 367.391,Z 473.667,A -85,B 0,C 180,E1 -12693.29,E2 -12693.29} C_VEL
LIN {X 0,Y 367.442,Z 471.155,A -85,B 0,C 180,E1 -12695.488,E2 -12695.488} C_VEL
LIN {X 0,Y 367.567,Z 467.368,A -85,B 0,C 180,E1 -12697.692,E2 -12697.692} C_VEL
LIN {X 0,Y 367.787,Z 462.217,A -85,B 0,C 180,E1 -12699.903,E2 -12699.903} C_VEL
LIN {X 0,Y 368.364,Z 455.572,A -85,B 0,C 180,E1 -12702.115,E2 -12702.115} C_VEL
LIN {X 0,Y 369.146,Z 447.219,A -85,B 0,C 180,E1 -12704.33,E2 -12704.33} C_VEL
LIN {X 0,Y 370.241,Z 438.25,A -85,B 0,C 180,E1 -12706.26,E2 -12706.26} C_VEL
LIN {X 0,Y 371.419,Z 429.059,A -85,B 0,C 180,E1 -12707.908,E2 -12707.908} C_VEL
LIN {X 0,Y 372.563,Z 419.231,A -85,B 0,C 180,E1 -12709.405,E2 -12709.405} C_VEL
LIN {X 0,Y 374,Z 407.362,A -85,B 0,C 180,E1 -12710.918,E2 -12710.918} C_VEL
LIN {X 0,Y 376.301,Z 392.194,A -85,B 0,C 180,E1 -12712.656,E2 -12712.656} C_VEL
LIN {X 0,Y 378.381,Z 378.277,A -85,B 0,C 180,E1 -12713.973,E2 -12713.973} C_VEL
LIN {X 0,Y 380.572,Z 362.46,A -85,B 0,C 180,E1 -12715.193,E2 -12715.193} C_VEL
LIN {X 0,Y 382.488,Z 347.564,A -85,B 0,C 180,E1 -12716.094,E2 -12716.094} C_VEL
LIN {X 0,Y 384.408,Z 330.896,A -85,B 0,C 180,E1 -12716.867,E2 -12716.867} C_VEL
LIN {X 0,Y 385.912,Z 312.318,A -85,B 0,C 180,E1 -12717.487,E2 -12717.487} C_VEL
LIN {X 0,Y 391.505,Z 239.18,A -85,B 0,C 180,E1 -12719.692,E2 -12719.692} C_VEL
LIN {X 0,Y 394.876,Z 200.955,A -85,B 0,C 180,E1 -12720.908,E2 -12720.908} C_VEL
LIN {X 0,Y 394.164,Z 181.122,A -85,B 0,C 180,E1 -12721.992,E2 -12721.992} C_VEL
LIN {X 0,Y 393.553,Z 172.116,A -85,B 0,C 180,E1 -12722.573,E2 -12722.573} C_VEL
LIN {X 0,Y 390.548,Z 161.931,A -85,B 0,C 180,E1 -12723.745,E2 -12723.745} C_VEL
LIN {X 0,Y 387.717,Z 152.499,A -85,B 0,C 180,E1 -12724.98,E2 -12724.98} C_VEL
LIN {X 0,Y 384.827,Z 148.219,A -85,B 0,C 180,E1 -12726.043,E2 -12726.043} C_VEL
LIN {X 0,Y 382.424,Z 144.876,A -85,B 0,C 180,E1 -12727.032,E2 -12727.032} C_VEL
LIN {X 0,Y 379.755,Z 141.032,A -85,B 0,C 180,E1 -12728.317,E2 -12728.317} C_VEL
LIN {X 0,Y 378.103,Z 139.328,A -85,B 0,C 180,E1 -12729.196,E2 -12729.196} C_VEL
LIN {X 0,Y 376.377,Z 135.902,A -85,B 0,C 180,E1 -12730.81,E2 -12730.81} C_VEL
LIN {X 0,Y 374.256,Z 134.174,A -85,B 0,C 180,E1 -12732.915,E2 -12732.915} C_VEL
LIN {X 0,Y 373.591,Z 133.309,A -85,B 0,C 180,E1 -12734.369,E2 -12734.369} C_VEL
LIN {X 0,Y 373.379,Z 132.99,A -85,B 0,C 180,E1 -12735.858,E2 -12735.858} C_VEL
LIN {X 0,Y 373.782,Z 133.807,A -85,B 0,C 180,E1 -12738.215,E2 -12738.215} C_VEL
LIN {X 0,Y 375.923,Z 135.837,A -85,B 0,C 180,E1 -12740.247,E2 -12740.247} C_VEL
LIN {X 0,Y 377.057,Z 137.227,A -85,B 0,C 180,E1 -12741.075,E2 -12741.075} C_VEL
LIN {X 0,Y 379.876,Z 140.621,A -85,B 0,C 180,E1 -12742.706,E2 -12742.706} C_VEL
LIN {X 0,Y 384.133,Z 146.495,A -85,B 0,C 180,E1 -12744.631,E2 -12744.631} C_VEL
LIN {X 0,Y 387.107,Z 150.88,A -85,B 0,C 180,E1 -12745.75,E2 -12745.75} C_VEL
LIN {X 0,Y 391.233,Z 157.511,A -85,B 0,C 180,E1 -12747.124,E2 -12747.124} C_VEL
LIN {X 0,Y 394.968,Z 164.163,A -85,B 0,C 180,E1 -12748.244,E2 -12748.244} C_VEL
LIN {X 0,Y 397.501,Z 169.523,A -85,B 0,C 180,E1 -12748.974,E2 -12748.974} C_VEL
LIN {X 0,Y 390.536,Z 245.222,A -85,B 0,C 180,E1 -12751.334,E2 -12751.334} C_VEL
LIN {X 0,Y 386.898,Z 294.163,A -85,B 0,C 180,E1 -12752.837,E2 -12752.837} C_VEL
LIN {X 0,Y 385.57,Z 309.955,A -85,B 0,C 180,E1 -12753.53,E2 -12753.53} C_VEL
LIN {X 0,Y 384.048,Z 324.628,A -85,B 0,C 180,E1 -12754.385,E2 -12754.385} C_VEL
LIN {X 0,Y 382.347,Z 338.838,A -85,B 0,C 180,E1 -12755.426,E2 -12755.426} C_VEL
LIN {X 0,Y 380.341,Z 353.328,A -85,B 0,C 180,E1 -12756.736,E2 -12756.736} C_VEL
LIN {X 0,Y 378.32,Z 366.98,A -85,B 0,C 180,E1 -12758.255,E2 -12758.255} C_VEL
LIN {X 0,Y 376.659,Z 376.649,A -85,B 0,C 180,E1 -12759.522,E2 -12759.522} C_VEL
LIN {X 0,Y 374.948,Z 387.05,A -85,B 0,C 180,E1 -12761.136,E2 -12761.136} C_VEL
LIN {X 0,Y 373.282,Z 397.208,A -85,B 0,C 180,E1 -12763.033,E2 -12763.033} C_VEL
LIN {X 0,Y 371.764,Z 405.68,A -85,B 0,C 180,E1 -12764.934,E2 -12764.934} C_VEL
LIN {X 0,Y 370.565,Z 412.712,A -85,B 0,C 180,E1 -12766.845,E2 -12766.845} C_VEL
LIN {X 0,Y 369.519,Z 419.169,A -85,B 0,C 180,E1 -12769.036,E2 -12769.036} C_VEL
LIN {X 0,Y 368.791,Z 424.138,A -85,B 0,C 180,E1 -12771.231,E2 -12771.231} C_VEL
LIN {X 0,Y 368.221,Z 427.756,A -85,B 0,C 180,E1 -12773.425,E2 -12773.425} C_VEL
LIN {X 0,Y 367.928,Z 430.079,A -85,B 0,C 180,E1 -12775.618,E2 -12775.618} C_VEL
LIN {X 0,Y 367.739,Z 431.158,A -85,B 0,C 180,E1 -12777.81,E2 -12777.81} C_VEL
LIN {X 0,Y 367.583,Z 430.974,A -85,B 0,C 180,E1 -12780,E2 -12780} C_VEL
LIN {X 0,Y 367.655,Z 429.532,A -85,B 0,C 180,E1 -12782.191,E2 -12782.191} C_VEL
LIN {X 0,Y 367.666,Z 426.829,A -85,B 0,C 180,E1 -12784.386,E2 -12784.386} C_VEL
LIN {X 0,Y 367.881,Z 422.794,A -85,B 0,C 180,E1 -12786.582,E2 -12786.582} C_VEL
LIN {X 0,Y 368.17,Z 417.339,A -85,B 0,C 180,E1 -12788.784,E2 -12788.784} C_VEL
LIN {X 0,Y 368.609,Z 410.319,A -85,B 0,C 180,E1 -12790.992,E2 -12790.992} C_VEL
LIN {X 0,Y 369.335,Z 402.7,A -85,B 0,C 180,E1 -12792.92,E2 -12792.92} C_VEL
LIN {X 0,Y 370.046,Z 393.492,A -85,B 0,C 180,E1 -12794.857,E2 -12794.857} C_VEL
LIN {X 0,Y 370.935,Z 384.081,A -85,B 0,C 180,E1 -12796.511,E2 -12796.511} C_VEL
LIN {X 0,Y 372.034,Z 372.963,A -85,B 0,C 180,E1 -12798.162,E2 -12798.162} C_VEL
LIN {X 0,Y 373.089,Z 361.198,A -85,B 0,C 180,E1 -12799.632,E2 -12799.632} C_VEL
LIN {X 0,Y 374.394,Z 347.647,A -85,B 0,C 180,E1 -12801.04,E2 -12801.04} C_VEL
LIN {X 0,Y 375.387,Z 334.912,A -85,B 0,C 180,E1 -12802.135,E2 -12802.135} C_VEL
LIN {X 0,Y 376.534,Z 320.352,A -85,B 0,C 180,E1 -12803.15,E2 -12803.15} C_VEL
LIN {X 0,Y 377.378,Z 305.262,A -85,B 0,C 180,E1 -12803.98,E2 -12803.98} C_VEL
LIN {X 0,Y 378.13,Z 289.345,A -85,B 0,C 180,E1 -12804.626,E2 -12804.626} C_VEL
LIN {X 0,Y 378.867,Z 267.012,A -85,B 0,C 180,E1 -12805.215,E2 -12805.215} C_VEL
LIN {X 0,Y 382.762,Z 157.996,A -85,B 0,C 180,E1 -12807.876,E2 -12807.876} C_VEL
LIN {X 0,Y 375.881,Z 141.811,A -85,B 0,C 180,E1 -12808.735,E2 -12808.735} C_VEL
LIN {X 0,Y 368.978,Z 125.642,A -85,B 0,C 180,E1 -12809.635,E2 -12809.635} C_VEL
LIN {X 0,Y 368.93,Z 125.157,A -85,B 0,C 180,E1 -12809.689,E2 -12809.689} C_VEL
LIN {X 0,Y 368.897,Z 125.161,A -85,B 0,C 180,E1 -12813.538,E2 -12813.538} C_VEL
LIN {X 0,Y 368.901,Z 125.157,A -85,B 0,C 180,E1 -12816.855,E2 -12816.855} C_VEL
LIN {X 0,Y 368.885,Z 125.158,A -85,B 0,C 180,E1 -12820.374,E2 -12820.374} C_VEL
LIN {X 0,Y 368.881,Z 125.156,A -85,B 0,C 180,E1 -12823.615,E2 -12823.615} C_VEL
LIN {X 0,Y 368.885,Z 125.133,A -85,B 0,C 180,E1 -12826.696,E2 -12826.696} C_VEL
LIN {X 0,Y 368.886,Z 125.16,A -85,B 0,C 180,E1 -12829.648,E2 -12829.648} C_VEL
LIN {X 0,Y 368.899,Z 125.143,A -85,B 0,C 180,E1 -12833.146,E2 -12833.146} C_VEL
LIN {X 0,Y 368.897,Z 125.153,A -85,B 0,C 180,E1 -12836.462,E2 -12836.462} C_VEL
LIN {X 0,Y 368.915,Z 125.15,A -85,B 0,C 180,E1 -12839.045,E2 -12839.045} C_VEL
LIN {X 0,Y 368.914,Z 125.148,A -85,B 0,C 180,E1 -12841.558,E2 -12841.558} C_VEL
LIN {X 0,Y 368.925,Z 125.154,A -85,B 0,C 180,E1 -12844.014,E2 -12844.014} C_VEL
LIN {X 0,Y 368.921,Z 125.154,A -85,B 0,C 180,E1 -12847.604,E2 -12847.604} C_VEL
LIN {X 0,Y 368.929,Z 125.152,A -85,B 0,C 180,E1 -12851.104,E2 -12851.104} C_VEL
LIN {X 0,Y 368.943,Z 125.149,A -85,B 0,C 180,E1 -12854.533,E2 -12854.533} C_VEL
LIN {X 0,Y 369.061,Z 125.134,A -85,B 0,C 180,E1 -12856.79,E2 -12856.79} C_VEL
LIN {X 0,Y 369.064,Z 125.135,A -85,B 0,C 180,E1 -12860.132,E2 -12860.132} C_VEL
LIN {X 0,Y 369.175,Z 125.307,A -85,B 0,C 180,E1 -12862.995,E2 -12862.995} C_VEL
LIN {X 0,Y 374.017,Z 142.613,A -85,B 0,C 180,E1 -12866.313,E2 -12866.313} C_VEL
LIN {X 0,Y 374.482,Z 144.182,A -85,B 0,C 180,E1 -12866.58,E2 -12866.58} C_VEL
LIN {X 0,Y 382.527,Z 163.377,A -85,B 0,C 180,E1 -12867.655,E2 -12867.655} C_VEL
LIN {X 0,Y 385.617,Z 178.257,A -85,B 0,C 180,E1 -12868.214,E2 -12868.214} C_VEL
LIN {X 0,Y 382.853,Z 291.303,A -85,B 0,C 180,E1 -12870.375,E2 -12870.375} C_VEL
LIN {X 0,Y 382.13,Z 297.15,A -85,B 0,C 180,E1 -12870.442,E2 -12870.442} C_VEL
LIN {X 0,Y 376.259,Z 316.098,A -85,B 0,C 180,E1 -12870.51,E2 -12870.51} C_VEL
LIN {X 0,Y 375.37,Z 321.859,A -85,B 0,C 180,E1 -12870.66,E2 -12870.66} C_VEL
LIN {X 0,Y 374.459,Z 336.297,A -85,B 0,C 180,E1 -12871.277,E2 -12871.277} C_VEL
LIN {X 0,Y 373.286,Z 350.487,A -85,B 0,C 180,E1 -12872.091,E2 -12872.091} C_VEL
LIN {X 0,Y 371.862,Z 364.341,A -85,B 0,C 180,E1 -12873.105,E2 -12873.105} C_VEL
LIN {X 0,Y 370.187,Z 378.03,A -85,B 0,C 180,E1 -12874.355,E2 -12874.355} C_VEL
LIN {X 0,Y 368.529,Z 391.189,A -85,B 0,C 180,E1 -12875.843,E2 -12875.843} C_VEL
LIN {X 0,Y 366.854,Z 402.799,A -85,B 0,C 180,E1 -12877.43,E2 -12877.43} C_VEL
LIN {X 0,Y 365.396,Z 413.131,A -85,B 0,C 180,E1 -12879.13,E2 -12879.13} C_VEL
LIN {X 0,Y 364.068,Z 422.099,A -85,B 0,C 180,E1 -12880.888,E2 -12880.888} C_VEL
LIN {X 0,Y 362.885,Z 430.53,A -85,B 0,C 180,E1 -12882.869,E2 -12882.869} C_VEL
LIN {X 0,Y 362.096,Z 436.737,A -85,B 0,C 180,E1 -12884.615,E2 -12884.615} C_VEL
LIN {X 0,Y 361.269,Z 443.502,A -85,B 0,C 180,E1 -12886.966,E2 -12886.966} C_VEL
LIN {X 0,Y 360.735,Z 448.737,A -85,B 0,C 180,E1 -12889.342,E2 -12889.342} C_VEL
LIN {X 0,Y 360.31,Z 452.564,A -85,B 0,C 180,E1 -12891.753,E2 -12891.753} C_VEL
LIN {X 0,Y 360.095,Z 455.001,A -85,B 0,C 180,E1 -12894.196,E2 -12894.196} C_VEL
LIN {X 0,Y 360.045,Z 456.057,A -85,B 0,C 180,E1 -12896.677,E2 -12896.677} C_VEL
LIN {X 0,Y 360.098,Z 455.947,A -85,B 0,C 180,E1 -12898.566,E2 -12898.566} C_VEL
LIN {X 0,Y 360.202,Z 454.695,A -85,B 0,C 180,E1 -12900.851,E2 -12900.851} C_VEL
LIN {X 0,Y 360.48,Z 452.275,A -85,B 0,C 180,E1 -12903.086,E2 -12903.086} C_VEL
LIN {X 0,Y 360.872,Z 449.028,A -85,B 0,C 180,E1 -12905.119,E2 -12905.119} C_VEL
LIN {X 0,Y 361.351,Z 444.842,A -85,B 0,C 180,E1 -12907.115,E2 -12907.115} C_VEL
LIN {X 0,Y 362.154,Z 438.72,A -85,B 0,C 180,E1 -12909.385,E2 -12909.385} C_VEL
LIN {X 0,Y 363.186,Z 431.526,A -85,B 0,C 180,E1 -12911.512,E2 -12911.512} C_VEL
LIN {X 0,Y 364.611,Z 422.789,A -85,B 0,C 180,E1 -12913.608,E2 -12913.608} C_VEL
LIN {X 0,Y 366,Z 414.49,A -85,B 0,C 180,E1 -12915.274,E2 -12915.274} C_VEL
LIN {X 0,Y 367.6,Z 404.312,A -85,B 0,C 180,E1 -12916.995,E2 -12916.995} C_VEL
LIN {X 0,Y 369.312,Z 393.368,A -85,B 0,C 180,E1 -12918.538,E2 -12918.538} C_VEL
LIN {X 0,Y 371.144,Z 380.882,A -85,B 0,C 180,E1 -12919.999,E2 -12919.999} C_VEL
LIN {X 0,Y 372.988,Z 366.892,A -85,B 0,C 180,E1 -12921.327,E2 -12921.327} C_VEL
LIN {X 0,Y 374.643,Z 352.32,A -85,B 0,C 180,E1 -12922.427,E2 -12922.427} C_VEL
LIN {X 0,Y 376.001,Z 338.032,A -85,B 0,C 180,E1 -12923.264,E2 -12923.264} C_VEL
LIN {X 0,Y 376.993,Z 323.498,A -85,B 0,C 180,E1 -12923.904,E2 -12923.904} C_VEL
LIN {X 0,Y 377.774,Z 307.722,A -85,B 0,C 180,E1 -12924.366,E2 -12924.366} C_VEL
LIN {X 0,Y 381.515,Z 174.331,A -85,B 0,C 180,E1 -12927.006,E2 -12927.006} C_VEL
LIN {X 0,Y 380.674,Z 170.039,A -85,B 0,C 180,E1 -12927.183,E2 -12927.183} C_VEL
LIN {X 0,Y 373.554,Z 153.972,A -85,B 0,C 180,E1 -12928.25,E2 -12928.25} C_VEL
LIN {X 0,Y 368.103,Z 143.219,A -85,B 0,C 180,E1 -12929.084,E2 -12929.084} C_VEL
LIN {X 0,Y 365.38,Z 135.522,A -85,B 0,C 180,E1 -12930.417,E2 -12930.417} C_VEL
LIN {X 0,Y 366.441,Z 136.936,A -85,B 0,C 180,E1 -12930.551,E2 -12930.551} C_VEL
LIN {X 0,Y 376.219,Z 159.444,A -85,B 0,C 180,E1 -12931.805,E2 -12931.805} C_VEL
LIN {X 0,Y 371.505,Z 287.799,A -85,B 0,C 180,E1 -12935.07,E2 -12935.07} C_VEL
LIN {X 0,Y 370.758,Z 303.149,A -85,B 0,C 180,E1 -12935.67,E2 -12935.67} C_VEL
LIN {X 0,Y 369.879,Z 318.341,A -85,B 0,C 180,E1 -12936.483,E2 -12936.483} C_VEL
LIN {X 0,Y 368.825,Z 332.519,A -85,B 0,C 180,E1 -12937.45,E2 -12937.45} C_VEL
LIN {X 0,Y 367.58,Z 347.196,A -85,B 0,C 180,E1 -12938.698,E2 -12938.698} C_VEL
LIN {X 0,Y 366.364,Z 360.202,A -85,B 0,C 180,E1 -12940.047,E2 -12940.047} C_VEL
LIN {X 0,Y 365.176,Z 372.857,A -85,B 0,C 180,E1 -12941.63,E2 -12941.63} C_VEL
LIN {X 0,Y 363.986,Z 384.959,A -85,B 0,C 180,E1 -12943.453,E2 -12943.453} C_VEL
LIN {X 0,Y 363.051,Z 394.331,A -85,B 0,C 180,E1 -12945.137,E2 -12945.137} C_VEL
LIN {X 0,Y 362.33,Z 403.522,A -85,B 0,C 180,E1 -12947.111,E2 -12947.111} C_VEL
LIN {X 0,Y 361.628,Z 410.155,A -85,B 0,C 180,E1 -12948.793,E2 -12948.793} C_VEL
LIN {X 0,Y 361.142,Z 417.379,A -85,B 0,C 180,E1 -12951.043,E2 -12951.043} C_VEL
LIN {X 0,Y 360.816,Z 423.012,A -85,B 0,C 180,E1 -12953.288,E2 -12953.288} C_VEL
LIN {X 0,Y 360.619,Z 427.208,A -85,B 0,C 180,E1 -12955.529,E2 -12955.529} C_VEL
LIN {X 0,Y 360.607,Z 430.074,A -85,B 0,C 180,E1 -12957.766,E2 -12957.766} C_VEL
LIN {X 0,Y 360.526,Z 431.659,A -85,B 0,C 180,E1 -12960,E2 -12960} C_VEL
LIN {X 0,Y 360.696,Z 431.973,A -85,B 0,C 180,E1 -12962.233,E2 -12962.233} C_VEL
LIN {X 0,Y 360.9,Z 431.054,A -85,B 0,C 180,E1 -12964.467,E2 -12964.467} C_VEL
LIN {X 0,Y 361.23,Z 428.901,A -85,B 0,C 180,E1 -12966.703,E2 -12966.703} C_VEL
LIN {X 0,Y 361.828,Z 425.462,A -85,B 0,C 180,E1 -12968.939,E2 -12968.939} C_VEL
LIN {X 0,Y 362.618,Z 420.692,A -85,B 0,C 180,E1 -12971.175,E2 -12971.175} C_VEL
LIN {X 0,Y 363.745,Z 414.453,A -85,B 0,C 180,E1 -12973.406,E2 -12973.406} C_VEL
LIN {X 0,Y 364.978,Z 407.683,A -85,B 0,C 180,E1 -12975.353,E2 -12975.353} C_VEL
LIN {X 0,Y 366.634,Z 399.477,A -85,B 0,C 180,E1 -12977.284,E2 -12977.284} C_VEL
LIN {X 0,Y 368.433,Z 389.632,A -85,B 0,C 180,E1 -12979.211,E2 -12979.211} C_VEL
LIN {X 0,Y 370.254,Z 379.616,A -85,B 0,C 180,E1 -12980.849,E2 -12980.849} C_VEL
LIN {X 0,Y 372.354,Z 367.951,A -85,B 0,C 180,E1 -12982.441,E2 -12982.441} C_VEL
LIN {X 0,Y 374.46,Z 354.764,A -85,B 0,C 180,E1 -12983.945,E2 -12983.945} C_VEL
LIN {X 0,Y 376.612,Z 340.512,A -85,B 0,C 180,E1 -12985.269,E2 -12985.269} C_VEL
LIN {X 0,Y 378.687,Z 324.71,A -85,B 0,C 180,E1 -12986.449,E2 -12986.449} C_VEL
LIN {X 0,Y 380.396,Z 309.603,A -85,B 0,C 180,E1 -12987.331,E2 -12987.331} C_VEL
LIN {X 0,Y 381.875,Z 293.708,A -85,B 0,C 180,E1 -12988.031,E2 -12988.031} C_VEL
LIN {X 0,Y 388.269,Z 220.155,A -85,B 0,C 180,E1 -12990.377,E2 -12990.377} C_VEL
LIN {X 0,Y 392.982,Z 175.303,A -85,B 0,C 180,E1 -12991.838,E2 -12991.838} C_VEL
LIN {X 0,Y 388.827,Z 167.536,A -85,B 0,C 180,E1 -12993.142,E2 -12993.142} C_VEL
LIN {X 0,Y 384.562,Z 160.793,A -85,B 0,C 180,E1 -12994.628,E2 -12994.628} C_VEL
LIN {X 0,Y 382.235,Z 157.425,A -85,B 0,C 180,E1 -12995.534,E2 -12995.534} C_VEL
LIN {X 0,Y 379.103,Z 153.467,A -85,B 0,C 180,E1 -12996.911,E2 -12996.911} C_VEL
LIN {X 0,Y 376.009,Z 149.742,A -85,B 0,C 180,E1 -12998.618,E2 -12998.618} C_VEL
LIN {X 0,Y 372.964,Z 146.69,A -85,B 0,C 180,E1 -13000.994,E2 -13000.994} C_VEL
LIN {X 0,Y 372.209,Z 146.11,A -85,B 0,C 180,E1 -13001.878,E2 -13001.878} C_VEL
LIN {X 0,Y 371.191,Z 146.009,A -85,B 0,C 180,E1 -13003.988,E2 -13003.988} C_VEL
LIN {X 0,Y 371.323,Z 147.089,A -85,B 0,C 180,E1 -13005.99,E2 -13005.99} C_VEL
LIN {X 0,Y 372.438,Z 149.401,A -85,B 0,C 180,E1 -13007.933,E2 -13007.933} C_VEL
LIN {X 0,Y 374.898,Z 153.22,A -85,B 0,C 180,E1 -13010.083,E2 -13010.083} C_VEL
LIN {X 0,Y 379.152,Z 160.853,A -85,B 0,C 180,E1 -13012.599,E2 -13012.599} C_VEL
LIN {X 0,Y 383.147,Z 168.705,A -85,B 0,C 180,E1 -13014.403,E2 -13014.403} C_VEL
LIN {X 0,Y 386.083,Z 175.348,A -85,B 0,C 180,E1 -13015.569,E2 -13015.569} C_VEL
LIN {X 0,Y 388.273,Z 180.643,A -85,B 0,C 180,E1 -13016.369,E2 -13016.369} C_VEL
LIN {X 0,Y 389.905,Z 195.502,A -85,B 0,C 180,E1 -13017.519,E2 -13017.519} C_VEL
LIN {X 0,Y 390.666,Z 207.758,A -85,B 0,C 180,E1 -13018.286,E2 -13018.286} C_VEL
LIN {X 0,Y 383.518,Z 284.953,A -85,B 0,C 180,E1 -13020.722,E2 -13020.722} C_VEL
LIN {X 0,Y 380.312,Z 325.319,A -85,B 0,C 180,E1 -13021.998,E2 -13021.998} C_VEL
LIN {X 0,Y 378.358,Z 341.809,A -85,B 0,C 180,E1 -13022.705,E2 -13022.705} C_VEL
LIN {X 0,Y 376.007,Z 358.817,A -85,B 0,C 180,E1 -13023.676,E2 -13023.676} C_VEL
LIN {X 0,Y 373.784,Z 373.719,A -85,B 0,C 180,E1 -13024.776,E2 -13024.776} C_VEL
LIN {X 0,Y 371.563,Z 387.345,A -85,B 0,C 180,E1 -13026.004,E2 -13026.004} C_VEL
LIN {X 0,Y 369.562,Z 399.73,A -85,B 0,C 180,E1 -13027.35,E2 -13027.35} C_VEL
LIN {X 0,Y 367.126,Z 415.192,A -85,B 0,C 180,E1 -13029.259,E2 -13029.259} C_VEL
LIN {X 0,Y 365.533,Z 426.406,A -85,B 0,C 180,E1 -13030.922,E2 -13030.922} C_VEL
LIN {X 0,Y 363.936,Z 437.285,A -85,B 0,C 180,E1 -13032.873,E2 -13032.873} C_VEL
LIN {X 0,Y 362.629,Z 446.303,A -85,B 0,C 180,E1 -13034.833,E2 -13034.833} C_VEL
LIN {X 0,Y 361.845,Z 452.768,A -85,B 0,C 180,E1 -13036.522,E2 -13036.522} C_VEL
LIN {X 0,Y 361.077,Z 459.92,A -85,B 0,C 180,E1 -13038.776,E2 -13038.776} C_VEL
LIN {X 0,Y 360.612,Z 465.53,A -85,B 0,C 180,E1 -13041.03,E2 -13041.03} C_VEL
LIN {X 0,Y 360.442,Z 469.748,A -85,B 0,C 180,E1 -13043.282,E2 -13043.282} C_VEL
LIN {X 0,Y 360.334,Z 472.681,A -85,B 0,C 180,E1 -13045.525,E2 -13045.525} C_VEL
LIN {X 0,Y 360.318,Z 474.397,A -85,B 0,C 180,E1 -13047.764,E2 -13047.764} C_VEL
LIN {X 0,Y 360.362,Z 474.926,A -85,B 0,C 180,E1 -13050,E2 -13050} C_VEL
LIN {X 0,Y 360.318,Z 474.261,A -85,B 0,C 180,E1 -13052.236,E2 -13052.236} C_VEL
LIN {X 0,Y 360.354,Z 472.358,A -85,B 0,C 180,E1 -13054.474,E2 -13054.474} C_VEL
LIN {X 0,Y 360.476,Z 469.204,A -85,B 0,C 180,E1 -13056.718,E2 -13056.718} C_VEL
LIN {X 0,Y 360.569,Z 464.729,A -85,B 0,C 180,E1 -13058.971,E2 -13058.971} C_VEL
LIN {X 0,Y 361.04,Z 458.832,A -85,B 0,C 180,E1 -13061.225,E2 -13061.225} C_VEL
LIN {X 0,Y 361.673,Z 451.335,A -85,B 0,C 180,E1 -13063.485,E2 -13063.485} C_VEL
LIN {X 0,Y 362.648,Z 443.248,A -85,B 0,C 180,E1 -13065.454,E2 -13065.454} C_VEL
LIN {X 0,Y 363.927,Z 433.489,A -85,B 0,C 180,E1 -13067.417,E2 -13067.417} C_VEL
LIN {X 0,Y 365.296,Z 422.44,A -85,B 0,C 180,E1 -13069.259,E2 -13069.259} C_VEL
LIN {X 0,Y 367.969,Z 404.733,A -85,B 0,C 180,E1 -13071.719,E2 -13071.719} C_VEL
LIN {X 0,Y 370.253,Z 390.775,A -85,B 0,C 180,E1 -13073.343,E2 -13073.343} C_VEL
LIN {X 0,Y 372.545,Z 376.385,A -85,B 0,C 180,E1 -13074.71,E2 -13074.71} C_VEL
LIN {X 0,Y 375,Z 360.003,A -85,B 0,C 180,E1 -13075.966,E2 -13075.966} C_VEL
LIN {X 0,Y 377.11,Z 344.871,A -85,B 0,C 180,E1 -13076.868,E2 -13076.868} C_VEL
LIN {X 0,Y 379.027,Z 328.291,A -85,B 0,C 180,E1 -13077.617,E2 -13077.617} C_VEL
LIN {X 0,Y 380.784,Z 307.687,A -85,B 0,C 180,E1 -13078.301,E2 -13078.301} C_VEL
LIN {X 0,Y 386.566,Z 238.889,A -85,B 0,C 180,E1 -13080.45,E2 -13080.45} C_VEL
LIN {X 0,Y 390.076,Z 202.217,A -85,B 0,C 180,E1 -13081.652,E2 -13081.652} C_VEL
LIN {X 0,Y 389.636,Z 183.515,A -85,B 0,C 180,E1 -13082.708,E2 -13082.708} C_VEL
LIN {X 0,Y 389.124,Z 175.226,A -85,B 0,C 180,E1 -13083.27,E2 -13083.27} C_VEL
LIN {X 0,Y 385.13,Z 160.454,A -85,B 0,C 180,E1 -13085.097,E2 -13085.097} C_VEL
LIN {X 0,Y 384.206,Z 157.68,A -85,B 0,C 180,E1 -13085.523,E2 -13085.523} C_VEL
LIN {X 0,Y 380.676,Z 152.18,A -85,B 0,C 180,E1 -13086.979,E2 -13086.979} C_VEL
LIN {X 0,Y 377.21,Z 147.301,A -85,B 0,C 180,E1 -13088.688,E2 -13088.688} C_VEL
LIN {X 0,Y 374.1,Z 143.006,A -85,B 0,C 180,E1 -13090.759,E2 -13090.759} C_VEL
LIN {X 0,Y 373.405,Z 142.183,A -85,B 0,C 180,E1 -13091.35,E2 -13091.35} C_VEL
LIN {X 0,Y 371.504,Z 140.363,A -85,B 0,C 180,E1 -13093.725,E2 -13093.725} C_VEL
LIN {X 0,Y 371.108,Z 139.748,A -85,B 0,C 180,E1 -13095.517,E2 -13095.517} C_VEL
LIN {X 0,Y 371.657,Z 140.271,A -85,B 0,C 180,E1 -13097.518,E2 -13097.518} C_VEL
LIN {X 0,Y 373.585,Z 142.202,A -85,B 0,C 180,E1 -13099.808,E2 -13099.808} C_VEL
LIN {X 0,Y 374.909,Z 143.777,A -85,B 0,C 180,E1 -13100.822,E2 -13100.822} C_VEL
LIN {X 0,Y 377.715,Z 147.289,A -85,B 0,C 180,E1 -13102.535,E2 -13102.535} C_VEL
LIN {X 0,Y 381.415,Z 152.68,A -85,B 0,C 180,E1 -13104.296,E2 -13104.296} C_VEL
LIN {X 0,Y 384.323,Z 157.223,A -85,B 0,C 180,E1 -13105.467,E2 -13105.467} C_VEL
LIN {X 0,Y 387.694,Z 162.811,A -85,B 0,C 180,E1 -13106.663,E2 -13106.663} C_VEL
LIN {X 0,Y 391.272,Z 169.466,A -85,B 0,C 180,E1 -13107.814,E2 -13107.814} C_VEL
LIN {X 0,Y 392.756,Z 172.789,A -85,B 0,C 180,E1 -13108.284,E2 -13108.284} C_VEL
LIN {X 0,Y 384.921,Z 251.664,A -85,B 0,C 180,E1 -13110.802,E2 -13110.802} C_VEL
LIN {X 0,Y 381.491,Z 294.343,A -85,B 0,C 180,E1 -13112.154,E2 -13112.154} C_VEL
LIN {X 0,Y 380.103,Z 309.329,A -85,B 0,C 180,E1 -13112.817,E2 -13112.817} C_VEL
LIN {X 0,Y 378.471,Z 324.192,A -85,B 0,C 180,E1 -13113.683,E2 -13113.683} C_VEL
LIN {X 0,Y 376.642,Z 338.5,A -85,B 0,C 180,E1 -13114.733,E2 -13114.733} C_VEL
LIN {X 0,Y 374.502,Z 353.03,A -85,B 0,C 180,E1 -13116.058,E2 -13116.058} C_VEL
LIN {X 0,Y 372.367,Z 366.455,A -85,B 0,C 180,E1 -13117.56,E2 -13117.56} C_VEL
LIN {X 0,Y 370.198,Z 378.328,A -85,B 0,C 180,E1 -13119.148,E2 -13119.148} C_VEL
LIN {X 0,Y 368.397,Z 388.506,A -85,B 0,C 180,E1 -13120.787,E2 -13120.787} C_VEL
LIN {X 0,Y 366.614,Z 398.482,A -85,B 0,C 180,E1 -13122.715,E2 -13122.715} C_VEL
LIN {X 0,Y 364.997,Z 406.801,A -85,B 0,C 180,E1 -13124.648,E2 -13124.648} C_VEL
LIN {X 0,Y 363.711,Z 413.695,A -85,B 0,C 180,E1 -13126.593,E2 -13126.593} C_VEL
LIN {X 0,Y 362.595,Z 420.032,A -85,B 0,C 180,E1 -13128.824,E2 -13128.824} C_VEL
LIN {X 0,Y 361.8,Z 424.891,A -85,B 0,C 180,E1 -13131.06,E2 -13131.06} C_VEL
LIN {X 0,Y 361.199,Z 428.403,A -85,B 0,C 180,E1 -13133.296,E2 -13133.296} C_VEL
LIN {X 0,Y 360.852,Z 430.629,A -85,B 0,C 180,E1 -13135.532,E2 -13135.532} C_VEL
LIN {X 0,Y 360.841,Z 431.27,A -85,B 0,C 180,E1 -13136.651,E2 -13136.651} C_VEL
LIN {X 0,Y 360.563,Z 431.644,A -85,B 0,C 180,E1 -13138.883,E2 -13138.883} C_VEL
LIN {X 0,Y 360.54,Z 430.747,A -85,B 0,C 180,E1 -13141.117,E2 -13141.117} C_VEL
LIN {X 0,Y 360.549,Z 428.58,A -85,B 0,C 180,E1 -13143.353,E2 -13143.353} C_VEL
LIN {X 0,Y 360.694,Z 425.109,A -85,B 0,C 180,E1 -13145.591,E2 -13145.591} C_VEL
LIN {X 0,Y 360.943,Z 420.264,A -85,B 0,C 180,E1 -13147.834,E2 -13147.834} C_VEL
LIN {X 0,Y 361.322,Z 413.92,A -85,B 0,C 180,E1 -13150.082,E2 -13150.082} C_VEL
LIN {X 0,Y 361.927,Z 406.962,A -85,B 0,C 180,E1 -13152.049,E2 -13152.049} C_VEL
LIN {X 0,Y 362.571,Z 398.224,A -85,B 0,C 180,E1 -13154.09,E2 -13154.09} C_VEL
LIN {X 0,Y 363.568,Z 388.379,A -85,B 0,C 180,E1 -13155.99,E2 -13155.99} C_VEL
LIN {X 0,Y 364.565,Z 377.956,A -85,B 0,C 180,E1 -13157.676,E2 -13157.676} C_VEL
LIN {X 0,Y 365.74,Z 366.279,A -85,B 0,C 180,E1 -13159.264,E2 -13159.264} C_VEL
LIN {X 0,Y 366.982,Z 353.215,A -85,B 0,C 180,E1 -13160.75,E2 -13160.75} C_VEL
LIN {X 0,Y 368.111,Z 339.884,A -85,B 0,C 180,E1 -13162.005,E2 -13162.005} C_VEL
LIN {X 0,Y 369.295,Z 325.388,A -85,B 0,C 180,E1 -13163.111,E2 -13163.111} C_VEL
LIN {X 0,Y 370.279,Z 310.32,A -85,B 0,C 180,E1 -13164.022,E2 -13164.022} C_VEL
LIN {X 0,Y 371.069,Z 294.698,A -85,B 0,C 180,E1 -13164.737,E2 -13164.737} C_VEL
LIN {X 0,Y 371.77,Z 277.211,A -85,B 0,C 180,E1 -13165.285,E2 -13165.285} C_VEL
LIN {X 0,Y 376.082,Z 159.485,A -85,B 0,C 180,E1 -13168.235,E2 -13168.235} C_VEL
LIN {X 0,Y 361.932,Z 126.456,A -85,B 0,C 180,E1 -13170.077,E2 -13170.077} C_VEL
LIN {X 0,Y 361.866,Z 126.036,A -85,B 0,C 180,E1 -13170.101,E2 -13170.101} C_VEL
LIN {X 0,Y 361.86,Z 126.036,A -85,B 0,C 180,E1 -13173.369,E2 -13173.369} C_VEL
LIN {X 0,Y 361.866,Z 126.034,A -85,B 0,C 180,E1 -13177.019,E2 -13177.019} C_VEL
LIN {X 0,Y 361.814,Z 126.04,A -85,B 0,C 180,E1 -13180.751,E2 -13180.751} C_VEL
LIN {X 0,Y 361.814,Z 126.033,A -85,B 0,C 180,E1 -13184.37,E2 -13184.37} C_VEL
LIN {X 0,Y 361.828,Z 126.017,A -85,B 0,C 180,E1 -13187.57,E2 -13187.57} C_VEL
LIN {X 0,Y 361.846,Z 126.034,A -85,B 0,C 180,E1 -13191.572,E2 -13191.572} C_VEL
LIN {X 0,Y 361.873,Z 126.012,A -85,B 0,C 180,E1 -13194.656,E2 -13194.656} C_VEL
LIN {X 0,Y 361.84,Z 126.037,A -85,B 0,C 180,E1 -13198.371,E2 -13198.371} C_VEL
LIN {X 0,Y 361.869,Z 126.02,A -85,B 0,C 180,E1 -13200.952,E2 -13200.952} C_VEL
LIN {X 0,Y 361.856,Z 126.029,A -85,B 0,C 180,E1 -13204.705,E2 -13204.705} C_VEL
LIN {X 0,Y 361.863,Z 126.036,A -85,B 0,C 180,E1 -13208.345,E2 -13208.345} C_VEL
LIN {X 0,Y 361.907,Z 126.03,A -85,B 0,C 180,E1 -13212.093,E2 -13212.093} C_VEL
LIN {X 0,Y 361.983,Z 126.02,A -85,B 0,C 180,E1 -13216.113,E2 -13216.113} C_VEL
LIN {X 0,Y 362.001,Z 126.014,A -85,B 0,C 180,E1 -13219.937,E2 -13219.937} C_VEL
LIN {X 0,Y 362.094,Z 126.077,A -85,B 0,C 180,E1 -13222.437,E2 -13222.437} C_VEL
LIN {X 0,Y 365.076,Z 136.422,A -85,B 0,C 180,E1 -13224.476,E2 -13224.476} C_VEL
LIN {X 0,Y 367.246,Z 144.39,A -85,B 0,C 180,E1 -13225.968,E2 -13225.968} C_VEL
LIN {X 0,Y 374.64,Z 161.189,A -85,B 0,C 180,E1 -13226.97,E2 -13226.97} C_VEL
LIN {X 0,Y 376.675,Z 166.771,A -85,B 0,C 180,E1 -13227.26,E2 -13227.26} C_VEL
LIN {X 0,Y 379.295,Z 179.337,A -85,B 0,C 180,E1 -13227.743,E2 -13227.743} C_VEL
LIN {X 0,Y 375.91,Z 311.239,A -85,B 0,C 180,E1 -13230.335,E2 -13230.335} C_VEL
LIN {X 0,Y 375.37,Z 321.859,A -85,B 0,C 180,E1 -13230.66,E2 -13230.66} C_VEL
LIN {X 0,Y 374.393,Z 327.589,A -85,B 0,C 180,E1 -13230.831,E2 -13230.831} C_VEL
LIN {X 0,Y 371.125,Z 336.832,A -85,B 0,C 180,E1 -13231.073,E2 -13231.073} C_VEL
LIN {X 0,Y 367.747,Z 345.941,A -85,B 0,C 180,E1 -13231.391,E2 -13231.391} C_VEL
LIN {X 0,Y 366.689,Z 351.365,A -85,B 0,C 180,E1 -13231.702,E2 -13231.702} C_VEL
LIN {X 0,Y 365.197,Z 365.368,A -85,B 0,C 180,E1 -13232.757,E2 -13232.757} C_VEL
LIN {X 0,Y 363.483,Z 378.821,A -85,B 0,C 180,E1 -13234.019,E2 -13234.019} C_VEL
LIN {X 0,Y 361.855,Z 391.088,A -85,B 0,C 180,E1 -13235.433,E2 -13235.433} C_VEL
LIN {X 0,Y 360.18,Z 402.449,A -85,B 0,C 180,E1 -13237.005,E2 -13237.005} C_VEL
LIN {X 0,Y 358.606,Z 412.887,A -85,B 0,C 180,E1 -13238.736,E2 -13238.736} C_VEL
LIN {X 0,Y 357.288,Z 421.406,A -85,B 0,C 180,E1 -13240.413,E2 -13240.413} C_VEL
LIN {X 0,Y 355.969,Z 430.417,A -85,B 0,C 180,E1 -13242.543,E2 -13242.543} C_VEL
LIN {X 0,Y 355.06,Z 437.138,A -85,B 0,C 180,E1 -13244.47,E2 -13244.47} C_VEL
LIN {X 0,Y 354.254,Z 443.494,A -85,B 0,C 180,E1 -13246.718,E2 -13246.718} C_VEL
LIN {X 0,Y 353.692,Z 448.774,A -85,B 0,C 180,E1 -13249.139,E2 -13249.139} C_VEL
LIN {X 0,Y 353.312,Z 451.836,A -85,B 0,C 180,E1 -13250.981,E2 -13250.981} C_VEL
LIN {X 0,Y 353.075,Z 454.663,A -85,B 0,C 180,E1 -13253.46,E2 -13253.46} C_VEL
LIN {X 0,Y 352.955,Z 456.12,A -85,B 0,C 180,E1 -13255.98,E2 -13255.98} C_VEL
LIN {X 0,Y 353.002,Z 456.163,A -85,B 0,C 180,E1 -13258.543,E2 -13258.543} C_VEL
LIN {X 0,Y 353.126,Z 454.702,A -85,B 0,C 180,E1 -13261.162,E2 -13261.162} C_VEL
LIN {X 0,Y 353.435,Z 452.303,A -85,B 0,C 180,E1 -13263.366,E2 -13263.366} C_VEL
LIN {X 0,Y 353.883,Z 448.896,A -85,B 0,C 180,E1 -13265.486,E2 -13265.486} C_VEL
LIN {X 0,Y 354.562,Z 443.658,A -85,B 0,C 180,E1 -13267.914,E2 -13267.914} C_VEL
LIN {X 0,Y 355.391,Z 437.745,A -85,B 0,C 180,E1 -13270.039,E2 -13270.039} C_VEL
LIN {X 0,Y 356.465,Z 430.717,A -85,B 0,C 180,E1 -13272.093,E2 -13272.093} C_VEL
LIN {X 0,Y 357.986,Z 421.98,A -85,B 0,C 180,E1 -13274.182,E2 -13274.182} C_VEL
LIN {X 0,Y 359.564,Z 412.987,A -85,B 0,C 180,E1 -13275.965,E2 -13275.965} C_VEL
LIN {X 0,Y 361.394,Z 401.573,A -85,B 0,C 180,E1 -13277.852,E2 -13277.852} C_VEL
LIN {X 0,Y 363.291,Z 390.155,A -85,B 0,C 180,E1 -13279.403,E2 -13279.403} C_VEL
LIN {X 0,Y 365.029,Z 378.571,A -85,B 0,C 180,E1 -13280.717,E2 -13280.717} C_VEL
LIN {X 0,Y 366.81,Z 365.212,A -85,B 0,C 180,E1 -13281.965,E2 -13281.965} C_VEL
LIN {X 0,Y 368.505,Z 350.667,A -85,B 0,C 180,E1 -13283.048,E2 -13283.048} C_VEL
LIN {X 0,Y 369.838,Z 336.735,A -85,B 0,C 180,E1 -13283.852,E2 -13283.852} C_VEL
LIN {X 0,Y 370.902,Z 321.755,A -85,B 0,C 180,E1 -13284.493,E2 -13284.493} C_VEL
LIN {X 0,Y 371.697,Z 305.362,A -85,B 0,C 180,E1 -13284.95,E2 -13284.95} C_VEL
LIN {X 0,Y 375.408,Z 174.856,A -85,B 0,C 180,E1 -13287.578,E2 -13287.578} C_VEL
LIN {X 0,Y 374.63,Z 172.049,A -85,B 0,C 180,E1 -13287.72,E2 -13287.72} C_VEL
LIN {X 0,Y 367.476,Z 156.058,A -85,B 0,C 180,E1 -13288.833,E2 -13288.833} C_VEL
LIN {X 0,Y 360.898,Z 143.389,A -85,B 0,C 180,E1 -13289.868,E2 -13289.868} C_VEL
LIN {X 0,Y 360.22,Z 141.303,A -85,B 0,C 180,E1 -13290.271,E2 -13290.271} C_VEL
LIN {X 0,Y 361.741,Z 143.221,A -85,B 0,C 180,E1 -13290.427,E2 -13290.427} C_VEL
LIN {X 0,Y 369.623,Z 161.346,A -85,B 0,C 180,E1 -13291.455,E2 -13291.455} C_VEL
LIN {X 0,Y 364.717,Z 288.169,A -85,B 0,C 180,E1 -13294.764,E2 -13294.764} C_VEL
LIN {X 0,Y 363.937,Z 303.401,A -85,B 0,C 180,E1 -13295.373,E2 -13295.373} C_VEL
LIN {X 0,Y 363.001,Z 319.149,A -85,B 0,C 180,E1 -13296.237,E2 -13296.237} C_VEL
LIN {X 0,Y 361.826,Z 334.094,A -85,B 0,C 180,E1 -13297.291,E2 -13297.291} C_VEL
LIN {X 0,Y 360.573,Z 348.553,A -85,B 0,C 180,E1 -13298.564,E2 -13298.564} C_VEL
LIN {X 0,Y 359.305,Z 361.893,A -85,B 0,C 180,E1 -13299.997,E2 -13299.997} C_VEL
LIN {X 0,Y 358.125,Z 373.928,A -85,B 0,C 180,E1 -13301.552,E2 -13301.552} C_VEL
LIN {X 0,Y 356.898,Z 385.932,A -85,B 0,C 180,E1 -13303.409,E2 -13303.409} C_VEL
LIN {X 0,Y 355.957,Z 395.221,A -85,B 0,C 180,E1 -13305.127,E2 -13305.127} C_VEL
LIN {X 0,Y 355.232,Z 404.343,A -85,B 0,C 180,E1 -13307.139,E2 -13307.139} C_VEL
LIN {X 0,Y 354.455,Z 411.882,A -85,B 0,C 180,E1 -13309.142,E2 -13309.142} C_VEL
LIN {X 0,Y 353.986,Z 418.852,A -85,B 0,C 180,E1 -13311.436,E2 -13311.436} C_VEL
LIN {X 0,Y 353.685,Z 423.755,A -85,B 0,C 180,E1 -13313.485,E2 -13313.485} C_VEL
LIN {X 0,Y 353.549,Z 427.384,A -85,B 0,C 180,E1 -13315.439,E2 -13315.439} C_VEL
LIN {X 0,Y 353.511,Z 430.338,A -85,B 0,C 180,E1 -13317.721,E2 -13317.721} C_VEL
LIN {X 0,Y 353.461,Z 432.015,A -85,B 0,C 180,E1 -13320,E2 -13320} C_VEL
LIN {X 0,Y 353.639,Z 432.437,A -85,B 0,C 180,E1 -13322.278,E2 -13322.278} C_VEL
LIN {X 0,Y 353.801,Z 432.18,A -85,B 0,C 180,E1 -13323.416,E2 -13323.416} C_VEL
LIN {X 0,Y 353.879,Z 430.772,A -85,B 0,C 180,E1 -13325.698,E2 -13325.698} C_VEL
LIN {X 0,Y 354.521,Z 428.083,A -85,B 0,C 180,E1 -13327.976,E2 -13327.976} C_VEL
LIN {X 0,Y 355.301,Z 424.095,A -85,B 0,C 180,E1 -13330.254,E2 -13330.254} C_VEL
LIN {X 0,Y 356.286,Z 418.746,A -85,B 0,C 180,E1 -13332.532,E2 -13332.532} C_VEL
LIN {X 0,Y 357.577,Z 411.88,A -85,B 0,C 180,E1 -13334.803,E2 -13334.803} C_VEL
LIN {X 0,Y 359.208,Z 404.452,A -85,B 0,C 180,E1 -13336.773,E2 -13336.773} C_VEL
LIN {X 0,Y 361.046,Z 395.528,A -85,B 0,C 180,E1 -13338.734,E2 -13338.734} C_VEL
LIN {X 0,Y 362.828,Z 386.513,A -85,B 0,C 180,E1 -13340.405,E2 -13340.405} C_VEL
LIN {X 0,Y 365.129,Z 374.956,A -85,B 0,C 180,E1 -13342.184,E2 -13342.184} C_VEL
LIN {X 0,Y 367.475,Z 362.058,A -85,B 0,C 180,E1 -13343.829,E2 -13343.829} C_VEL
LIN {X 0,Y 369.663,Z 349.291,A -85,B 0,C 180,E1 -13345.175,E2 -13345.175} C_VEL
LIN {X 0,Y 371.743,Z 335.536,A -85,B 0,C 180,E1 -13346.377,E2 -13346.377} C_VEL
LIN {X 0,Y 373.788,Z 320.136,A -85,B 0,C 180,E1 -13347.46,E2 -13347.46} C_VEL
LIN {X 0,Y 375.682,Z 303.829,A -85,B 0,C 180,E1 -13348.34,E2 -13348.34} C_VEL
LIN {X 0,Y 377.149,Z 287.689,A -85,B 0,C 180,E1 -13348.979,E2 -13348.979} C_VEL
LIN {X 0,Y 383.551,Z 221.16,A -85,B 0,C 180,E1 -13351.151,E2 -13351.151} C_VEL
LIN {X 0,Y 388.344,Z 178.625,A -85,B 0,C 180,E1 -13352.578,E2 -13352.578} C_VEL
LIN {X 0,Y 384.545,Z 171.583,A -85,B 0,C 180,E1 -13353.881,E2 -13353.881} C_VEL
LIN {X 0,Y 381.008,Z 165.897,A -85,B 0,C 180,E1 -13355.236,E2 -13355.236} C_VEL
LIN {X 0,Y 378.95,Z 162.94,A -85,B 0,C 180,E1 -13356.106,E2 -13356.106} C_VEL
LIN {X 0,Y 376.589,Z 159.793,A -85,B 0,C 180,E1 -13357.237,E2 -13357.237} C_VEL
LIN {X 0,Y 373.798,Z 156.359,A -85,B 0,C 180,E1 -13358.864,E2 -13358.864} C_VEL
LIN {X 0,Y 370.868,Z 153.193,A -85,B 0,C 180,E1 -13361.391,E2 -13361.391} C_VEL
LIN {X 0,Y 369.49,Z 152.853,A -85,B 0,C 180,E1 -13363.715,E2 -13363.715} C_VEL
LIN {X 0,Y 369.495,Z 153.834,A -85,B 0,C 180,E1 -13365.795,E2 -13365.795} C_VEL
LIN {X 0,Y 370.467,Z 156.079,A -85,B 0,C 180,E1 -13367.719,E2 -13367.719} C_VEL
LIN {X 0,Y 372.759,Z 159.897,A -85,B 0,C 180,E1 -13369.873,E2 -13369.873} C_VEL
LIN {X 0,Y 376.694,Z 167.467,A -85,B 0,C 180,E1 -13372.358,E2 -13372.358} C_VEL
LIN {X 0,Y 380.008,Z 174.342,A -85,B 0,C 180,E1 -13373.959,E2 -13373.959} C_VEL
LIN {X 0,Y 382.508,Z 180.316,A -85,B 0,C 180,E1 -13375.038,E2 -13375.038} C_VEL
LIN {X 0,Y 384.238,Z 184.75,A -85,B 0,C 180,E1 -13375.735,E2 -13375.735} C_VEL
LIN {X 0,Y 385.557,Z 199.166,A -85,B 0,C 180,E1 -13376.877,E2 -13376.877} C_VEL
LIN {X 0,Y 386.001,Z 209.293,A -85,B 0,C 180,E1 -13377.521,E2 -13377.521} C_VEL
LIN {X 0,Y 378.685,Z 282.04,A -85,B 0,C 180,E1 -13379.889,E2 -13379.889} C_VEL
LIN {X 0,Y 374.978,Z 324.207,A -85,B 0,C 180,E1 -13381.258,E2 -13381.258} C_VEL
LIN {X 0,Y 372.779,Z 341.816,A -85,B 0,C 180,E1 -13382.033,E2 -13382.033} C_VEL
LIN {X 0,Y 370.511,Z 357.079,A -85,B 0,C 180,E1 -13382.919,E2 -13382.919} C_VEL
LIN {X 0,Y 368.233,Z 371.274,A -85,B 0,C 180,E1 -13383.962,E2 -13383.962} C_VEL
LIN {X 0,Y 365.686,Z 386.061,A -85,B 0,C 180,E1 -13385.291,E2 -13385.291} C_VEL
LIN {X 0,Y 363.271,Z 399.649,A -85,B 0,C 180,E1 -13386.785,E2 -13386.785} C_VEL
LIN {X 0,Y 360.295,Z 416.209,A -85,B 0,C 180,E1 -13388.996,E2 -13388.996} C_VEL
LIN {X 0,Y 358.79,Z 426.42,A -85,B 0,C 180,E1 -13390.549,E2 -13390.549} C_VEL
LIN {X 0,Y 357.089,Z 437.243,A -85,B 0,C 180,E1 -13392.534,E2 -13392.534} C_VEL
LIN {X 0,Y 355.728,Z 446.223,A -85,B 0,C 180,E1 -13394.531,E2 -13394.531} C_VEL
LIN {X 0,Y 354.618,Z 454.616,A -85,B 0,C 180,E1 -13396.826,E2 -13396.826} C_VEL
LIN {X 0,Y 353.885,Z 461.344,A -85,B 0,C 180,E1 -13399.125,E2 -13399.125} C_VEL
LIN {X 0,Y 353.473,Z 466.586,A -85,B 0,C 180,E1 -13401.424,E2 -13401.424} C_VEL
LIN {X 0,Y 353.361,Z 469.603,A -85,B 0,C 180,E1 -13403.146,E2 -13403.146} C_VEL
LIN {X 0,Y 353.247,Z 472.521,A -85,B 0,C 180,E1 -13405.435,E2 -13405.435} C_VEL
LIN {X 0,Y 353.222,Z 474.222,A -85,B 0,C 180,E1 -13407.719,E2 -13407.719} C_VEL
LIN {X 0,Y 353.264,Z 474.735,A -85,B 0,C 180,E1 -13410,E2 -13410} C_VEL
LIN {X 0,Y 353.222,Z 474.057,A -85,B 0,C 180,E1 -13412.281,E2 -13412.281} C_VEL
LIN {X 0,Y 353.265,Z 472.144,A -85,B 0,C 180,E1 -13414.564,E2 -13414.564} C_VEL
LIN {X 0,Y 353.382,Z 468.97,A -85,B 0,C 180,E1 -13416.853,E2 -13416.853} C_VEL
LIN {X 0,Y 353.512,Z 464.475,A -85,B 0,C 180,E1 -13419.151,E2 -13419.151} C_VEL
LIN {X 0,Y 353.997,Z 458.556,A -85,B 0,C 180,E1 -13421.451,E2 -13421.451} C_VEL
LIN {X 0,Y 354.672,Z 451.034,A -85,B 0,C 180,E1 -13423.756,E2 -13423.756} C_VEL
LIN {X 0,Y 355.712,Z 442.921,A -85,B 0,C 180,E1 -13425.763,E2 -13425.763} C_VEL
LIN {X 0,Y 357.081,Z 433.135,A -85,B 0,C 180,E1 -13427.762,E2 -13427.762} C_VEL
LIN {X 0,Y 359.466,Z 416.257,A -85,B 0,C 180,E1 -13430.605,E2 -13430.605} C_VEL
LIN {X 0,Y 361.668,Z 404.629,A -85,B 0,C 180,E1 -13432.267,E2 -13432.267} C_VEL
LIN {X 0,Y 363.852,Z 392.039,A -85,B 0,C 180,E1 -13433.779,E2 -13433.779} C_VEL
LIN {X 0,Y 366.296,Z 377.935,A -85,B 0,C 180,E1 -13435.185,E2 -13435.185} C_VEL
LIN {X 0,Y 368.88,Z 361.997,A -85,B 0,C 180,E1 -13436.46,E2 -13436.46} C_VEL
LIN {X 0,Y 371.308,Z 345.922,A -85,B 0,C 180,E1 -13437.475,E2 -13437.475} C_VEL
LIN {X 0,Y 373.415,Z 329.65,A -85,B 0,C 180,E1 -13438.259,E2 -13438.259} C_VEL
LIN {X 0,Y 375.28,Z 309.962,A -85,B 0,C 180,E1 -13438.946,E2 -13438.946} C_VEL
LIN {X 0,Y 381.69,Z 239.749,A -85,B 0,C 180,E1 -13441.208,E2 -13441.208} C_VEL
LIN {X 0,Y 385.449,Z 203.567,A -85,B 0,C 180,E1 -13442.424,E2 -13442.424} C_VEL
LIN {X 0,Y 385.274,Z 186.08,A -85,B 0,C 180,E1 -13443.446,E2 -13443.446} C_VEL
LIN {X 0,Y 384.93,Z 178.643,A -85,B 0,C 180,E1 -13443.97,E2 -13443.97} C_VEL
LIN {X 0,Y 381.541,Z 164.903,A -85,B 0,C 180,E1 -13445.73,E2 -13445.73} C_VEL
LIN {X 0,Y 380.826,Z 162.812,A -85,B 0,C 180,E1 -13446.088,E2 -13446.088} C_VEL
LIN {X 0,Y 377.397,Z 157.623,A -85,B 0,C 180,E1 -13447.595,E2 -13447.595} C_VEL
LIN {X 0,Y 374.797,Z 153.668,A -85,B 0,C 180,E1 -13449.017,E2 -13449.017} C_VEL
LIN {X 0,Y 372.024,Z 149.591,A -85,B 0,C 180,E1 -13451.013,E2 -13451.013} C_VEL
LIN {X 0,Y 371.015,Z 148.555,A -85,B 0,C 180,E1 -13451.937,E2 -13451.937} C_VEL
LIN {X 0,Y 369.578,Z 146.966,A -85,B 0,C 180,E1 -13454.203,E2 -13454.203} C_VEL
LIN {X 0,Y 369.426,Z 146.69,A -85,B 0,C 180,E1 -13456.296,E2 -13456.296} C_VEL
LIN {X 0,Y 370.448,Z 147.781,A -85,B 0,C 180,E1 -13458.394,E2 -13458.394} C_VEL
LIN {X 0,Y 372.419,Z 149.762,A -85,B 0,C 180,E1 -13460.286,E2 -13460.286} C_VEL
LIN {X 0,Y 375.102,Z 153.472,A -85,B 0,C 180,E1 -13462.107,E2 -13462.107} C_VEL
LIN {X 0,Y 376.78,Z 156.116,A -85,B 0,C 180,E1 -13463.043,E2 -13463.043} C_VEL
LIN {X 0,Y 378.615,Z 158.664,A -85,B 0,C 180,E1 -13463.91,E2 -13463.91} C_VEL
LIN {X 0,Y 381.258,Z 162.952,A -85,B 0,C 180,E1 -13465.047,E2 -13465.047} C_VEL
LIN {X 0,Y 384.623,Z 168.938,A -85,B 0,C 180,E1 -13466.342,E2 -13466.342} C_VEL
LIN {X 0,Y 387.769,Z 175.08,A -85,B 0,C 180,E1 -13467.417,E2 -13467.417} C_VEL
LIN {X 0,Y 388.097,Z 176.264,A -85,B 0,C 180,E1 -13467.555,E2 -13467.555} C_VEL
LIN {X 0,Y 379.553,Z 256.607,A -85,B 0,C 180,E1 -13470.195,E2 -13470.195} C_VEL
LIN {X 0,Y 376.158,Z 295.342,A -85,B 0,C 180,E1 -13471.463,E2 -13471.463} C_VEL
LIN {X 0,Y 374.608,Z 310.557,A -85,B 0,C 180,E1 -13472.16,E2 -13472.16} C_VEL
LIN {X 0,Y 372.753,Z 326.052,A -85,B 0,C 180,E1 -13473.096,E2 -13473.096} C_VEL
LIN {X 0,Y 370.801,Z 339.95,A -85,B 0,C 180,E1 -13474.156,E2 -13474.156} C_VEL
LIN {X 0,Y 368.549,Z 354.205,A -85,B 0,C 180,E1 -13475.496,E2 -13475.496} C_VEL
LIN {X 0,Y 366.42,Z 366.582,A -85,B 0,C 180,E1 -13476.907,E2 -13476.907} C_VEL
LIN {X 0,Y 364.129,Z 378.29,A -85,B 0,C 180,E1 -13478.487,E2 -13478.487} C_VEL
LIN {X 0,Y 361.87,Z 390.056,A -85,B 0,C 180,E1 -13480.427,E2 -13480.427} C_VEL
LIN {X 0,Y 359.97,Z 399.832,A -85,B 0,C 180,E1 -13482.385,E2 -13482.385} C_VEL
LIN {X 0,Y 358.268,Z 407.981,A -85,B 0,C 180,E1 -13484.352,E2 -13484.352} C_VEL
LIN {X 0,Y 356.867,Z 414.729,A -85,B 0,C 180,E1 -13486.331,E2 -13486.331} C_VEL
LIN {X 0,Y 355.68,Z 420.933,A -85,B 0,C 180,E1 -13488.604,E2 -13488.604} C_VEL
LIN {X 0,Y 354.826,Z 425.671,A -85,B 0,C 180,E1 -13490.883,E2 -13490.883} C_VEL
LIN {X 0,Y 354.176,Z 429.068,A -85,B 0,C 180,E1 -13493.163,E2 -13493.163} C_VEL
LIN {X 0,Y 353.779,Z 431.19,A -85,B 0,C 180,E1 -13495.443,E2 -13495.443} C_VEL
LIN {X 0,Y 353.768,Z 431.775,A -85,B 0,C 180,E1 -13496.584,E2 -13496.584} C_VEL
LIN {X 0,Y 353.501,Z 432.041,A -85,B 0,C 180,E1 -13498.861,E2 -13498.861} C_VEL
LIN {X 0,Y 353.459,Z 431.05,A -85,B 0,C 180,E1 -13501.14,E2 -13501.14} C_VEL
LIN {X 0,Y 353.46,Z 428.795,A -85,B 0,C 180,E1 -13503.42,E2 -13503.42} C_VEL
LIN {X 0,Y 353.607,Z 425.219,A -85,B 0,C 180,E1 -13505.704,E2 -13505.704} C_VEL
LIN {X 0,Y 353.878,Z 420.243,A -85,B 0,C 180,E1 -13507.991,E2 -13507.991} C_VEL
LIN {X 0,Y 354.283,Z 413.741,A -85,B 0,C 180,E1 -13510.285,E2 -13510.285} C_VEL
LIN {X 0,Y 354.925,Z 406.659,A -85,B 0,C 180,E1 -13512.291,E2 -13512.291} C_VEL
LIN {X 0,Y 355.607,Z 397.409,A -85,B 0,C 180,E1 -13514.441,E2 -13514.441} C_VEL
LIN {X 0,Y 356.628,Z 387.686,A -85,B 0,C 180,E1 -13516.31,E2 -13516.31} C_VEL
LIN {X 0,Y 357.689,Z 377.064,A -85,B 0,C 180,E1 -13518.027,E2 -13518.027} C_VEL
LIN {X 0,Y 358.873,Z 365.448,A -85,B 0,C 180,E1 -13519.607,E2 -13519.607} C_VEL
LIN {X 0,Y 360.227,Z 351.698,A -85,B 0,C 180,E1 -13521.158,E2 -13521.158} C_VEL
LIN {X 0,Y 361.41,Z 337.964,A -85,B 0,C 180,E1 -13522.435,E2 -13522.435} C_VEL
LIN {X 0,Y 362.627,Z 322.927,A -85,B 0,C 180,E1 -13523.562,E2 -13523.562} C_VEL
LIN {X 0,Y 363.605,Z 307.538,A -85,B 0,C 180,E1 -13524.468,E2 -13524.468} C_VEL
LIN {X 0,Y 364.411,Z 292.179,A -85,B 0,C 180,E1 -13525.144,E2 -13525.144} C_VEL
LIN {X 0,Y 365.082,Z 274.84,A -85,B 0,C 180,E1 -13525.667,E2 -13525.667} C_VEL
LIN {X 0,Y 369.442,Z 161.291,A -85,B 0,C 180,E1 -13528.588,E2 -13528.588} C_VEL
LIN {X 0,Y 354.998,Z 127.777,A -85,B 0,C 180,E1 -13530.509,E2 -13530.509} C_VEL
LIN {X 0,Y 354.828,Z 126.912,A -85,B 0,C 180,E1 -13530.574,E2 -13530.574} C_VEL
LIN {X 0,Y 354.808,Z 126.915,A -85,B 0,C 180,E1 -13533.702,E2 -13533.702} C_VEL
LIN {X 0,Y 354.797,Z 126.913,A -85,B 0,C 180,E1 -13536.46,E2 -13536.46} C_VEL
LIN {X 0,Y 354.77,Z 126.92,A -85,B 0,C 180,E1 -13539.413,E2 -13539.413} C_VEL
LIN {X 0,Y 354.786,Z 126.916,A -85,B 0,C 180,E1 -13542.867,E2 -13542.867} C_VEL
LIN {X 0,Y 354.764,Z 126.892,A -85,B 0,C 180,E1 -13546.103,E2 -13546.103} C_VEL
LIN {X 0,Y 354.766,Z 126.912,A -85,B 0,C 180,E1 -13549.176,E2 -13549.176} C_VEL
LIN {X 0,Y 354.802,Z 126.91,A -85,B 0,C 180,E1 -13552.404,E2 -13552.404} C_VEL
LIN {X 0,Y 354.81,Z 126.893,A -85,B 0,C 180,E1 -13554.941,E2 -13554.941} C_VEL
LIN {X 0,Y 354.796,Z 126.915,A -85,B 0,C 180,E1 -13558.405,E2 -13558.405} C_VEL
LIN {X 0,Y 354.802,Z 126.906,A -85,B 0,C 180,E1 -13561.615,E2 -13561.615} C_VEL
LIN {X 0,Y 354.805,Z 126.901,A -85,B 0,C 180,E1 -13565.42,E2 -13565.42} C_VEL
LIN {X 0,Y 354.827,Z 126.906,A -85,B 0,C 180,E1 -13569.113,E2 -13569.113} C_VEL
LIN {X 0,Y 354.854,Z 126.906,A -85,B 0,C 180,E1 -13572.718,E2 -13572.718} C_VEL
LIN {X 0,Y 354.943,Z 126.895,A -85,B 0,C 180,E1 -13576.255,E2 -13576.255} C_VEL
LIN {X 0,Y 354.957,Z 126.89,A -85,B 0,C 180,E1 -13579.735,E2 -13579.735} C_VEL
LIN {X 0,Y 355.082,Z 127.075,A -85,B 0,C 180,E1 -13581.907,E2 -13581.907} C_VEL
LIN {X 0,Y 358.669,Z 139.422,A -85,B 0,C 180,E1 -13584.378,E2 -13584.378} C_VEL
LIN {X 0,Y 359.884,Z 144.239,A -85,B 0,C 180,E1 -13585.307,E2 -13585.307} C_VEL
LIN {X 0,Y 365.985,Z 157.603,A -85,B 0,C 180,E1 -13586.16,E2 -13586.16} C_VEL
LIN {X 0,Y 370.688,Z 169.316,A -85,B 0,C 180,E1 -13586.824,E2 -13586.824} C_VEL
LIN {X 0,Y 372.988,Z 181.065,A -85,B 0,C 180,E1 -13587.276,E2 -13587.276} C_VEL
LIN {X 0,Y 369.491,Z 311.032,A -85,B 0,C 180,E1 -13589.864,E2 -13589.864} C_VEL
LIN {X 0,Y 368.649,Z 326.534,A -85,B 0,C 180,E1 -13590.375,E2 -13590.375} C_VEL
LIN {X 0,Y 367.609,Z 341.446,A -85,B 0,C 180,E1 -13591.095,E2 -13591.095} C_VEL
LIN {X 0,Y 366.689,Z 351.365,A -85,B 0,C 180,E1 -13591.702,E2 -13591.702} C_VEL
LIN {X 0,Y 365.562,Z 356.761,A -85,B 0,C 180,E1 -13592.036,E2 -13592.036} C_VEL
LIN {X 0,Y 361.945,Z 365.421,A -85,B 0,C 180,E1 -13592.545,E2 -13592.545} C_VEL
LIN {X 0,Y 358.211,Z 373.879,A -85,B 0,C 180,E1 -13593.131,E2 -13593.131} C_VEL
LIN {X 0,Y 356.884,Z 378.817,A -85,B 0,C 180,E1 -13593.594,E2 -13593.594} C_VEL
LIN {X 0,Y 355.103,Z 391.739,A -85,B 0,C 180,E1 -13595.11,E2 -13595.11} C_VEL
LIN {X 0,Y 353.533,Z 402.077,A -85,B 0,C 180,E1 -13596.565,E2 -13596.565} C_VEL
LIN {X 0,Y 351.856,Z 412.616,A -85,B 0,C 180,E1 -13598.326,E2 -13598.326} C_VEL
LIN {X 0,Y 350.203,Z 422.908,A -85,B 0,C 180,E1 -13600.406,E2 -13600.406} C_VEL
LIN {X 0,Y 348.905,Z 431.428,A -85,B 0,C 180,E1 -13602.506,E2 -13602.506} C_VEL
LIN {X 0,Y 347.884,Z 438.605,A -85,B 0,C 180,E1 -13604.672,E2 -13604.672} C_VEL
LIN {X 0,Y 347.091,Z 444.947,A -85,B 0,C 180,E1 -13607.074,E2 -13607.074} C_VEL
LIN {X 0,Y 346.522,Z 449.929,A -85,B 0,C 180,E1 -13609.551,E2 -13609.551} C_VEL
LIN {X 0,Y 346.145,Z 452.734,A -85,B 0,C 180,E1 -13611.436,E2 -13611.436} C_VEL
LIN {X 0,Y 345.937,Z 455.257,A -85,B 0,C 180,E1 -13613.974,E2 -13613.974} C_VEL
LIN {X 0,Y 345.856,Z 456.412,A -85,B 0,C 180,E1 -13616.605,E2 -13616.605} C_VEL
LIN {X 0,Y 345.93,Z 456.128,A -85,B 0,C 180,E1 -13619.182,E2 -13619.182} C_VEL
LIN {X 0,Y 346.094,Z 454.342,A -85,B 0,C 180,E1 -13621.869,E2 -13621.869} C_VEL
LIN {X 0,Y 346.427,Z 452.231,A -85,B 0,C 180,E1 -13623.718,E2 -13623.718} C_VEL
LIN {X 0,Y 346.909,Z 448.578,A -85,B 0,C 180,E1 -13625.98,E2 -13625.98} C_VEL
LIN {X 0,Y 347.622,Z 443.518,A -85,B 0,C 180,E1 -13628.31,E2 -13628.31} C_VEL
LIN {X 0,Y 348.758,Z 436.154,A -85,B 0,C 180,E1 -13630.914,E2 -13630.914} C_VEL
LIN {X 0,Y 350.052,Z 428.568,A -85,B 0,C 180,E1 -13633.049,E2 -13633.049} C_VEL
LIN {X 0,Y 351.731,Z 419.276,A -85,B 0,C 180,E1 -13635.181,E2 -13635.181} C_VEL
LIN {X 0,Y 353.569,Z 408.91,A -85,B 0,C 180,E1 -13637.137,E2 -13637.137} C_VEL
LIN {X 0,Y 355.516,Z 397.692,A -85,B 0,C 180,E1 -13638.888,E2 -13638.888} C_VEL
LIN {X 0,Y 357.569,Z 385.393,A -85,B 0,C 180,E1 -13640.471,E2 -13640.471} C_VEL
LIN {X 0,Y 359.577,Z 372.023,A -85,B 0,C 180,E1 -13641.878,E2 -13641.878} C_VEL
LIN {X 0,Y 361.314,Z 358.766,A -85,B 0,C 180,E1 -13643.008,E2 -13643.008} C_VEL
LIN {X 0,Y 362.863,Z 344.683,A -85,B 0,C 180,E1 -13643.962,E2 -13643.962} C_VEL
LIN {X 0,Y 364.237,Z 329.133,A -85,B 0,C 180,E1 -13644.753,E2 -13644.753} C_VEL
LIN {X 0,Y 365.216,Z 313.609,A -85,B 0,C 180,E1 -13645.299,E2 -13645.299} C_VEL
LIN {X 0,Y 366.42,Z 275.383,A -85,B 0,C 180,E1 -13646.116,E2 -13646.116} C_VEL
LIN {X 0,Y 369.444,Z 176.068,A -85,B 0,C 180,E1 -13648.147,E2 -13648.147} C_VEL
LIN {X 0,Y 362.86,Z 161.107,A -85,B 0,C 180,E1 -13649.206,E2 -13649.206} C_VEL
LIN {X 0,Y 356.633,Z 148.699,A -85,B 0,C 180,E1 -13650.255,E2 -13650.255} C_VEL
LIN {X 0,Y 362.838,Z 162.873,A -85,B 0,C 180,E1 -13651.075,E2 -13651.075} C_VEL
LIN {X 0,Y 357.915,Z 288.108,A -85,B 0,C 180,E1 -13654.443,E2 -13654.443} C_VEL
LIN {X 0,Y 357.102,Z 304.031,A -85,B 0,C 180,E1 -13655.095,E2 -13655.095} C_VEL
LIN {X 0,Y 356.088,Z 319.779,A -85,B 0,C 180,E1 -13655.979,E2 -13655.979} C_VEL
LIN {X 0,Y 354.99,Z 333.789,A -85,B 0,C 180,E1 -13656.982,E2 -13656.982} C_VEL
LIN {X 0,Y 353.684,Z 348.366,A -85,B 0,C 180,E1 -13658.278,E2 -13658.278} C_VEL
LIN {X 0,Y 352.386,Z 361.883,A -85,B 0,C 180,E1 -13659.748,E2 -13659.748} C_VEL
LIN {X 0,Y 351.157,Z 373.936,A -85,B 0,C 180,E1 -13661.323,E2 -13661.323} C_VEL
LIN {X 0,Y 349.999,Z 385.158,A -85,B 0,C 180,E1 -13663.072,E2 -13663.072} C_VEL
LIN {X 0,Y 349,Z 394.647,A -85,B 0,C 180,E1 -13664.823,E2 -13664.823} C_VEL
LIN {X 0,Y 348.234,Z 403.949,A -85,B 0,C 180,E1 -13666.876,E2 -13666.876} C_VEL
LIN {X 0,Y 347.428,Z 411.644,A -85,B 0,C 180,E1 -13668.92,E2 -13668.92} C_VEL
LIN {X 0,Y 346.924,Z 418.758,A -85,B 0,C 180,E1 -13671.261,E2 -13671.261} C_VEL
LIN {X 0,Y 346.617,Z 424.044,A -85,B 0,C 180,E1 -13673.476,E2 -13673.476} C_VEL
LIN {X 0,Y 346.481,Z 427.504,A -85,B 0,C 180,E1 -13675.346,E2 -13675.346} C_VEL
LIN {X 0,Y 346.415,Z 430.574,A -85,B 0,C 180,E1 -13677.674,E2 -13677.674} C_VEL
LIN {X 0,Y 346.397,Z 432.366,A -85,B 0,C 180,E1 -13680,E2 -13680} C_VEL
LIN {X 0,Y 346.584,Z 432.904,A -85,B 0,C 180,E1 -13682.324,E2 -13682.324} C_VEL
LIN {X 0,Y 346.757,Z 432.215,A -85,B 0,C 180,E1 -13684.65,E2 -13684.65} C_VEL
LIN {X 0,Y 347.199,Z 430.282,A -85,B 0,C 180,E1 -13686.976,E2 -13686.976} C_VEL
LIN {X 0,Y 347.877,Z 427.088,A -85,B 0,C 180,E1 -13689.301,E2 -13689.301} C_VEL
LIN {X 0,Y 348.78,Z 422.57,A -85,B 0,C 180,E1 -13691.624,E2 -13691.624} C_VEL
LIN {X 0,Y 350.101,Z 416.607,A -85,B 0,C 180,E1 -13693.939,E2 -13693.939} C_VEL
LIN {X 0,Y 351.54,Z 410.113,A -85,B 0,C 180,E1 -13695.955,E2 -13695.955} C_VEL
LIN {X 0,Y 353.613,Z 401.006,A -85,B 0,C 180,E1 -13698.242,E2 -13698.242} C_VEL
LIN {X 0,Y 355.748,Z 391.33,A -85,B 0,C 180,E1 -13700.226,E2 -13700.226} C_VEL
LIN {X 0,Y 357.822,Z 381.533,A -85,B 0,C 180,E1 -13701.912,E2 -13701.912} C_VEL
LIN {X 0,Y 360.362,Z 369.389,A -85,B 0,C 180,E1 -13703.641,E2 -13703.641} C_VEL
LIN {X 0,Y 362.616,Z 357.37,A -85,B 0,C 180,E1 -13705.085,E2 -13705.085} C_VEL
LIN {X 0,Y 365.041,Z 343.684,A -85,B 0,C 180,E1 -13706.437,E2 -13706.437} C_VEL
LIN {X 0,Y 367.345,Z 328.803,A -85,B 0,C 180,E1 -13707.635,E2 -13707.635} C_VEL
LIN {X 0,Y 369.496,Z 313.112,A -85,B 0,C 180,E1 -13708.627,E2 -13708.627} C_VEL
LIN {X 0,Y 371.239,Z 297.609,A -85,B 0,C 180,E1 -13709.379,E2 -13709.379} C_VEL
LIN {X 0,Y 373.754,Z 270.958,A -85,B 0,C 180,E1 -13710.315,E2 -13710.315} C_VEL
LIN {X 0,Y 381.619,Z 200.933,A -85,B 0,C 180,E1 -13712.678,E2 -13712.678} C_VEL
LIN {X 0,Y 383.913,Z 182.179,A -85,B 0,C 180,E1 -13713.334,E2 -13713.334} C_VEL
LIN {X 0,Y 380.589,Z 175.941,A -85,B 0,C 180,E1 -13714.588,E2 -13714.588} C_VEL
LIN {X 0,Y 377.099,Z 170.124,A -85,B 0,C 180,E1 -13716.088,E2 -13716.088} C_VEL
LIN {X 0,Y 373.937,Z 165.884,A -85,B 0,C 180,E1 -13717.667,E2 -13717.667} C_VEL
LIN {X 0,Y 371.724,Z 163.042,A -85,B 0,C 180,E1 -13719.05,E2 -13719.05} C_VEL
LIN {X 0,Y 368.893,Z 159.908,A -85,B 0,C 180,E1 -13721.657,E2 -13721.657} C_VEL
LIN {X 0,Y 367.662,Z 159.819,A -85,B 0,C 180,E1 -13724.138,E2 -13724.138} C_VEL
LIN {X 0,Y 367.881,Z 161.167,A -85,B 0,C 180,E1 -13726.243,E2 -13726.243} C_VEL
LIN {X 0,Y 369.231,Z 164.098,A -85,B 0,C 180,E1 -13728.37,E2 -13728.37} C_VEL
LIN {X 0,Y 370.57,Z 166.518,A -85,B 0,C 180,E1 -13729.614,E2 -13729.614} C_VEL
LIN {X 0,Y 374.032,Z 173.585,A -85,B 0,C 180,E1 -13731.979,E2 -13731.979} C_VEL
LIN {X 0,Y 376.915,Z 179.99,A -85,B 0,C 180,E1 -13733.495,E2 -13733.495} C_VEL
LIN {X 0,Y 379.352,Z 186.189,A -85,B 0,C 180,E1 -13734.642,E2 -13734.642} C_VEL
LIN {X 0,Y 380.381,Z 189.138,A -85,B 0,C 180,E1 -13735.11,E2 -13735.11} C_VEL
LIN {X 0,Y 381.356,Z 203.857,A -85,B 0,C 180,E1 -13736.275,E2 -13736.275} C_VEL
LIN {X 0,Y 381.452,Z 211.229,A -85,B 0,C 180,E1 -13736.735,E2 -13736.735} C_VEL
LIN {X 0,Y 373.489,Z 284.663,A -85,B 0,C 180,E1 -13739.191,E2 -13739.191} C_VEL
LIN {X 0,Y 369.684,Z 324.499,A -85,B 0,C 180,E1 -13740.534,E2 -13740.534} C_VEL
LIN {X 0,Y 367.273,Z 342.215,A -85,B 0,C 180,E1 -13741.342,E2 -13741.342} C_VEL
LIN {X 0,Y 364.737,Z 358.058,A -85,B 0,C 180,E1 -13742.299,E2 -13742.299} C_VEL
LIN {X 0,Y 362.044,Z 373.417,A -85,B 0,C 180,E1 -13743.482,E2 -13743.482} C_VEL
LIN {X 0,Y 359.372,Z 387.605,A -85,B 0,C 180,E1 -13744.827,E2 -13744.827} C_VEL
LIN {X 0,Y 356.854,Z 400.764,A -85,B 0,C 180,E1 -13746.342,E2 -13746.342} C_VEL
LIN {X 0,Y 354.223,Z 413.905,A -85,B 0,C 180,E1 -13748.16,E2 -13748.16} C_VEL
LIN {X 0,Y 351.499,Z 429.689,A -85,B 0,C 180,E1 -13750.737,E2 -13750.737} C_VEL
LIN {X 0,Y 350.04,Z 438.57,A -85,B 0,C 180,E1 -13752.472,E2 -13752.472} C_VEL
LIN {X 0,Y 348.635,Z 447.288,A -85,B 0,C 180,E1 -13754.508,E2 -13754.508} C_VEL
LIN {X 0,Y 347.643,Z 454.529,A -85,B 0,C 180,E1 -13756.557,E2 -13756.557} C_VEL
LIN {X 0,Y 346.851,Z 461.228,A -85,B 0,C 180,E1 -13758.902,E2 -13758.902} C_VEL
LIN {X 0,Y 346.414,Z 466.449,A -85,B 0,C 180,E1 -13761.248,E2 -13761.248} C_VEL
LIN {X 0,Y 346.263,Z 469.459,A -85,B 0,C 180,E1 -13763.005,E2 -13763.005} C_VEL
LIN {X 0,Y 346.146,Z 472.362,A -85,B 0,C 180,E1 -13765.342,E2 -13765.342} C_VEL
LIN {X 0,Y 346.129,Z 474.048,A -85,B 0,C 180,E1 -13767.673,E2 -13767.673} C_VEL
LIN {X 0,Y 346.167,Z 474.545,A -85,B 0,C 180,E1 -13770,E2 -13770} C_VEL
LIN {X 0,Y 346.13,Z 473.851,A -85,B 0,C 180,E1 -13772.327,E2 -13772.327} C_VEL
LIN {X 0,Y 346.162,Z 471.928,A -85,B 0,C 180,E1 -13774.658,E2 -13774.658} C_VEL
LIN {X 0,Y 346.299,Z 468.736,A -85,B 0,C 180,E1 -13776.994,E2 -13776.994} C_VEL
LIN {X 0,Y 346.429,Z 464.219,A -85,B 0,C 180,E1 -13779.34,E2 -13779.34} C_VEL
LIN {X 0,Y 346.967,Z 458.28,A -85,B 0,C 180,E1 -13781.686,E2 -13781.686} C_VEL
LIN {X 0,Y 347.688,Z 450.734,A -85,B 0,C 180,E1 -13784.038,E2 -13784.038} C_VEL
LIN {X 0,Y 348.806,Z 442.596,A -85,B 0,C 180,E1 -13786.084,E2 -13786.084} C_VEL
LIN {X 0,Y 350.234,Z 432.779,A -85,B 0,C 180,E1 -13788.121,E2 -13788.121} C_VEL
LIN {X 0,Y 352.559,Z 419.147,A -85,B 0,C 180,E1 -13790.648,E2 -13790.648} C_VEL
LIN {X 0,Y 354.523,Z 408.618,A -85,B 0,C 180,E1 -13792.28,E2 -13792.28} C_VEL
LIN {X 0,Y 357,Z 395.819,A -85,B 0,C 180,E1 -13793.956,E2 -13793.956} C_VEL
LIN {X 0,Y 359.682,Z 381.756,A -85,B 0,C 180,E1 -13795.459,E2 -13795.459} C_VEL
LIN {X 0,Y 362.41,Z 366.543,A -85,B 0,C 180,E1 -13796.799,E2 -13796.799} C_VEL
LIN {X 0,Y 364.896,Z 351.587,A -85,B 0,C 180,E1 -13797.844,E2 -13797.844} C_VEL
LIN {X 0,Y 367.415,Z 334.594,A -85,B 0,C 180,E1 -13798.763,E2 -13798.763} C_VEL
LIN {X 0,Y 369.453,Z 317.477,A -85,B 0,C 180,E1 -13799.447,E2 -13799.447} C_VEL
LIN {X 0,Y 376.938,Z 241.221,A -85,B 0,C 180,E1 -13801.981,E2 -13801.981} C_VEL
LIN {X 0,Y 381.003,Z 204.808,A -85,B 0,C 180,E1 -13803.238,E2 -13803.238} C_VEL
LIN {X 0,Y 381.07,Z 187.195,A -85,B 0,C 180,E1 -13804.309,E2 -13804.309} C_VEL
LIN {X 0,Y 380.875,Z 181.944,A -85,B 0,C 180,E1 -13804.705,E2 -13804.705} C_VEL
LIN {X 0,Y 377.905,Z 168.754,A -85,B 0,C 180,E1 -13806.477,E2 -13806.477} C_VEL
LIN {X 0,Y 374.857,Z 163.871,A -85,B 0,C 180,E1 -13807.935,E2 -13807.935} C_VEL
LIN {X 0,Y 372.477,Z 160.128,A -85,B 0,C 180,E1 -13809.322,E2 -13809.322} C_VEL
LIN {X 0,Y 369.75,Z 155.838,A -85,B 0,C 180,E1 -13811.497,E2 -13811.497} C_VEL
LIN {X 0,Y 367.929,Z 153.994,A -85,B 0,C 180,E1 -13813.939,E2 -13813.939} C_VEL
LIN {X 0,Y 367.635,Z 153.6,A -85,B 0,C 180,E1 -13815.017,E2 -13815.017} C_VEL
LIN {X 0,Y 368.014,Z 153.886,A -85,B 0,C 180,E1 -13817.211,E2 -13817.211} C_VEL
LIN {X 0,Y 369.737,Z 155.685,A -85,B 0,C 180,E1 -13819.493,E2 -13819.493} C_VEL
LIN {X 0,Y 370.79,Z 157.165,A -85,B 0,C 180,E1 -13820.439,E2 -13820.439} C_VEL
LIN {X 0,Y 373.511,Z 161.002,A -85,B 0,C 180,E1 -13822.268,E2 -13822.268} C_VEL
LIN {X 0,Y 375.968,Z 164.998,A -85,B 0,C 180,E1 -13823.601,E2 -13823.601} C_VEL
LIN {X 0,Y 378.762,Z 169.709,A -85,B 0,C 180,E1 -13824.862,E2 -13824.862} C_VEL
LIN {X 0,Y 382.595,Z 176.907,A -85,B 0,C 180,E1 -13826.375,E2 -13826.375} C_VEL
LIN {X 0,Y 383.65,Z 179.232,A -85,B 0,C 180,E1 -13826.768,E2 -13826.768} C_VEL
LIN {X 0,Y 374.974,Z 254.765,A -85,B 0,C 180,E1 -13829.326,E2 -13829.326} C_VEL
LIN {X 0,Y 371.032,Z 295.562,A -85,B 0,C 180,E1 -13830.704,E2 -13830.704} C_VEL
LIN {X 0,Y 369.25,Z 312.081,A -85,B 0,C 180,E1 -13831.482,E2 -13831.482} C_VEL
LIN {X 0,Y 367.117,Z 328.108,A -85,B 0,C 180,E1 -13832.495,E2 -13832.495} C_VEL
LIN {X 0,Y 365.041,Z 341.605,A -85,B 0,C 180,E1 -13833.563,E2 -13833.563} C_VEL
LIN {X 0,Y 362.653,Z 355.568,A -85,B 0,C 180,E1 -13834.918,E2 -13834.918} C_VEL
LIN {X 0,Y 360.087,Z 369.254,A -85,B 0,C 180,E1 -13836.538,E2 -13836.538} C_VEL
LIN {X 0,Y 357.775,Z 380.201,A -85,B 0,C 180,E1 -13838.085,E2 -13838.085} C_VEL
LIN {X 0,Y 355.655,Z 390.174,A -85,B 0,C 180,E1 -13839.769,E2 -13839.769} C_VEL
LIN {X 0,Y 353.648,Z 399.96,A -85,B 0,C 180,E1 -13841.76,E2 -13841.76} C_VEL
LIN {X 0,Y 351.568,Z 409.221,A -85,B 0,C 180,E1 -13844.046,E2 -13844.046} C_VEL
LIN {X 0,Y 350.048,Z 415.812,A -85,B 0,C 180,E1 -13846.059,E2 -13846.059} C_VEL
LIN {X 0,Y 348.774,Z 421.872,A -85,B 0,C 180,E1 -13848.375,E2 -13848.375} C_VEL
LIN {X 0,Y 347.865,Z 426.479,A -85,B 0,C 180,E1 -13850.699,E2 -13850.699} C_VEL
LIN {X 0,Y 347.142,Z 429.753,A -85,B 0,C 180,E1 -13853.023,E2 -13853.023} C_VEL
LIN {X 0,Y 346.709,Z 431.761,A -85,B 0,C 180,E1 -13855.35,E2 -13855.35} C_VEL
LIN {X 0,Y 346.571,Z 432.516,A -85,B 0,C 180,E1 -13857.676,E2 -13857.676} C_VEL
LIN {X 0,Y 346.389,Z 432.041,A -85,B 0,C 180,E1 -13860,E2 -13860} C_VEL
LIN {X 0,Y 346.369,Z 430.308,A -85,B 0,C 180,E1 -13862.326,E2 -13862.326} C_VEL
LIN {X 0,Y 346.461,Z 427.285,A -85,B 0,C 180,E1 -13864.654,E2 -13864.654} C_VEL
LIN {X 0,Y 346.699,Z 422.894,A -85,B 0,C 180,E1 -13866.986,E2 -13866.986} C_VEL
LIN {X 0,Y 347.008,Z 417.03,A -85,B 0,C 180,E1 -13869.325,E2 -13869.325} C_VEL
LIN {X 0,Y 347.555,Z 409.528,A -85,B 0,C 180,E1 -13871.667,E2 -13871.667} C_VEL
LIN {X 0,Y 348.184,Z 402.732,A -85,B 0,C 180,E1 -13873.423,E2 -13873.423} C_VEL
LIN {X 0,Y 349.069,Z 393.225,A -85,B 0,C 180,E1 -13875.473,E2 -13875.473} C_VEL
LIN {X 0,Y 350.063,Z 383.53,A -85,B 0,C 180,E1 -13877.226,E2 -13877.226} C_VEL
LIN {X 0,Y 351.284,Z 372.042,A -85,B 0,C 180,E1 -13878.972,E2 -13878.972} C_VEL
LIN {X 0,Y 352.511,Z 359.417,A -85,B 0,C 180,E1 -13880.576,E2 -13880.576} C_VEL
LIN {X 0,Y 353.869,Z 345.685,A -85,B 0,C 180,E1 -13882.016,E2 -13882.016} C_VEL
LIN {X 0,Y 355.02,Z 332.368,A -85,B 0,C 180,E1 -13883.17,E2 -13883.17} C_VEL
LIN {X 0,Y 356.173,Z 318.059,A -85,B 0,C 180,E1 -13884.17,E2 -13884.17} C_VEL
LIN {X 0,Y 357.112,Z 302.147,A -85,B 0,C 180,E1 -13885.037,E2 -13885.037} C_VEL
LIN {X 0,Y 357.877,Z 285.905,A -85,B 0,C 180,E1 -13885.675,E2 -13885.675} C_VEL
LIN {X 0,Y 362.744,Z 162.926,A -85,B 0,C 180,E1 -13888.957,E2 -13888.957} C_VEL
LIN {X 0,Y 347.87,Z 128.449,A -85,B 0,C 180,E1 -13890.982,E2 -13890.982} C_VEL
LIN {X 0,Y 347.763,Z 127.792,A -85,B 0,C 180,E1 -13891.019,E2 -13891.019} C_VEL
LIN {X 0,Y 347.746,Z 127.792,A -85,B 0,C 180,E1 -13894.464,E2 -13894.464} C_VEL
LIN {X 0,Y 347.764,Z 127.791,A -85,B 0,C 180,E1 -13897.987,E2 -13897.987} C_VEL
LIN {X 0,Y 347.745,Z 127.794,A -85,B 0,C 180,E1 -13901.832,E2 -13901.832} C_VEL
LIN {X 0,Y 347.702,Z 127.781,A -85,B 0,C 180,E1 -13905.028,E2 -13905.028} C_VEL
LIN {X 0,Y 347.741,Z 127.781,A -85,B 0,C 180,E1 -13908.4,E2 -13908.4} C_VEL
LIN {X 0,Y 347.765,Z 127.786,A -85,B 0,C 180,E1 -13912.014,E2 -13912.014} C_VEL
LIN {X 0,Y 347.745,Z 127.779,A -85,B 0,C 180,E1 -13915.536,E2 -13915.536} C_VEL
LIN {X 0,Y 347.747,Z 127.792,A -85,B 0,C 180,E1 -13918.301,E2 -13918.301} C_VEL
LIN {X 0,Y 347.747,Z 127.778,A -85,B 0,C 180,E1 -13920.985,E2 -13920.985} C_VEL
LIN {X 0,Y 347.744,Z 127.793,A -85,B 0,C 180,E1 -13923.601,E2 -13923.601} C_VEL
LIN {X 0,Y 347.754,Z 127.778,A -85,B 0,C 180,E1 -13926.159,E2 -13926.159} C_VEL
LIN {X 0,Y 347.781,Z 127.78,A -85,B 0,C 180,E1 -13929.907,E2 -13929.907} C_VEL
LIN {X 0,Y 347.8,Z 127.779,A -85,B 0,C 180,E1 -13933.567,E2 -13933.567} C_VEL
LIN {X 0,Y 347.89,Z 127.77,A -85,B 0,C 180,E1 -13937.161,E2 -13937.161} C_VEL
LIN {X 0,Y 347.996,Z 127.826,A -85,B 0,C 180,E1 -13941.288,E2 -13941.288} C_VEL
LIN {X 0,Y 351.87,Z 140.971,A -85,B 0,C 180,E1 -13943.981,E2 -13943.981} C_VEL
LIN {X 0,Y 352.76,Z 144.478,A -85,B 0,C 180,E1 -13944.653,E2 -13944.653} C_VEL
LIN {X 0,Y 359.752,Z 159.588,A -85,B 0,C 180,E1 -13945.655,E2 -13945.655} C_VEL
LIN {X 0,Y 364.726,Z 171.989,A -85,B 0,C 180,E1 -13946.38,E2 -13946.38} C_VEL
LIN {X 0,Y 366.706,Z 182.086,A -85,B 0,C 180,E1 -13946.778,E2 -13946.778} C_VEL
LIN {X 0,Y 363.125,Z 310.611,A -85,B 0,C 180,E1 -13949.376,E2 -13949.376} C_VEL
LIN {X 0,Y 362.229,Z 326.353,A -85,B 0,C 180,E1 -13949.896,E2 -13949.896} C_VEL
LIN {X 0,Y 361.158,Z 341.351,A -85,B 0,C 180,E1 -13950.627,E2 -13950.627} C_VEL
LIN {X 0,Y 359.787,Z 355.168,A -85,B 0,C 180,E1 -13951.509,E2 -13951.509} C_VEL
LIN {X 0,Y 358.26,Z 368.794,A -85,B 0,C 180,E1 -13952.616,E2 -13952.616} C_VEL
LIN {X 0,Y 356.884,Z 378.817,A -85,B 0,C 180,E1 -13953.594,E2 -13953.594} C_VEL
LIN {X 0,Y 355.565,Z 383.714,A -85,B 0,C 180,E1 -13954.085,E2 -13954.085} C_VEL
LIN {X 0,Y 351.744,Z 391.502,A -85,B 0,C 180,E1 -13954.868,E2 -13954.868} C_VEL
LIN {X 0,Y 347.934,Z 398.99,A -85,B 0,C 180,E1 -13955.732,E2 -13955.732} C_VEL
LIN {X 0,Y 346.611,Z 403.302,A -85,B 0,C 180,E1 -13956.356,E2 -13956.356} C_VEL
LIN {X 0,Y 344.859,Z 413.941,A -85,B 0,C 180,E1 -13958.202,E2 -13958.202} C_VEL
LIN {X 0,Y 343.166,Z 423.97,A -85,B 0,C 180,E1 -13960.304,E2 -13960.304} C_VEL
LIN {X 0,Y 341.853,Z 432.41,A -85,B 0,C 180,E1 -13962.466,E2 -13962.466} C_VEL
LIN {X 0,Y 340.724,Z 440.036,A -85,B 0,C 180,E1 -13964.88,E2 -13964.88} C_VEL
LIN {X 0,Y 339.901,Z 446.174,A -85,B 0,C 180,E1 -13967.367,E2 -13967.367} C_VEL
LIN {X 0,Y 339.475,Z 449.958,A -85,B 0,C 180,E1 -13969.344,E2 -13969.344} C_VEL
LIN {X 0,Y 338.983,Z 453.588,A -85,B 0,C 180,E1 -13971.912,E2 -13971.912} C_VEL
LIN {X 0,Y 338.804,Z 455.82,A -85,B 0,C 180,E1 -13974.511,E2 -13974.511} C_VEL
LIN {X 0,Y 338.755,Z 456.674,A -85,B 0,C 180,E1 -13977.157,E2 -13977.157} C_VEL
LIN {X 0,Y 338.827,Z 456.263,A -85,B 0,C 180,E1 -13979.404,E2 -13979.404} C_VEL
LIN {X 0,Y 339.001,Z 454.727,A -85,B 0,C 180,E1 -13981.788,E2 -13981.788} C_VEL
LIN {X 0,Y 339.415,Z 452.151,A -85,B 0,C 180,E1 -13984.08,E2 -13984.08} C_VEL
LIN {X 0,Y 339.881,Z 448.685,A -85,B 0,C 180,E1 -13986.25,E2 -13986.25} C_VEL
LIN {X 0,Y 340.552,Z 444.233,A -85,B 0,C 180,E1 -13988.352,E2 -13988.352} C_VEL
LIN {X 0,Y 341.615,Z 437.922,A -85,B 0,C 180,E1 -13990.713,E2 -13990.713} C_VEL
LIN {X 0,Y 342.878,Z 430.426,A -85,B 0,C 180,E1 -13992.963,E2 -13992.963} C_VEL
LIN {X 0,Y 344.387,Z 422.722,A -85,B 0,C 180,E1 -13994.864,E2 -13994.864} C_VEL
LIN {X 0,Y 346.318,Z 412.637,A -85,B 0,C 180,E1 -13996.934,E2 -13996.934} C_VEL
LIN {X 0,Y 348.203,Z 401.971,A -85,B 0,C 180,E1 -13998.75,E2 -13998.75} C_VEL
LIN {X 0,Y 350.323,Z 390.44,A -85,B 0,C 180,E1 -14000.367,E2 -14000.367} C_VEL
LIN {X 0,Y 352.366,Z 378.038,A -85,B 0,C 180,E1 -14001.807,E2 -14001.807} C_VEL
LIN {X 0,Y 354.37,Z 364.161,A -85,B 0,C 180,E1 -14003.119,E2 -14003.119} C_VEL
LIN {X 0,Y 356.031,Z 350.502,A -85,B 0,C 180,E1 -14004.152,E2 -14004.152} C_VEL
LIN {X 0,Y 357.549,Z 335.474,A -85,B 0,C 180,E1 -14005.026,E2 -14005.026} C_VEL
LIN {X 0,Y 358.705,Z 320.515,A -85,B 0,C 180,E1 -14005.654,E2 -14005.654} C_VEL
LIN {X 0,Y 359.483,Z 304.531,A -85,B 0,C 180,E1 -14006.096,E2 -14006.096} C_VEL
LIN {X 0,Y 363.489,Z 178.12,A -85,B 0,C 180,E1 -14008.721,E2 -14008.721} C_VEL
LIN {X 0,Y 356.913,Z 163.279,A -85,B 0,C 180,E1 -14009.818,E2 -14009.818} C_VEL
LIN {X 0,Y 354.989,Z 159.803,A -85,B 0,C 180,E1 -14010.129,E2 -14010.129} C_VEL
LIN {X 0,Y 353.545,Z 158.505,A -85,B 0,C 180,E1 -14010.332,E2 -14010.332} C_VEL
LIN {X 0,Y 356.25,Z 164.863,A -85,B 0,C 180,E1 -14010.72,E2 -14010.72} C_VEL
LIN {X 0,Y 351.066,Z 288.871,A -85,B 0,C 180,E1 -14014.144,E2 -14014.144} C_VEL
LIN {X 0,Y 350.237,Z 304.547,A -85,B 0,C 180,E1 -14014.806,E2 -14014.806} C_VEL
LIN {X 0,Y 349.205,Z 320.284,A -85,B 0,C 180,E1 -14015.712,E2 -14015.712} C_VEL
LIN {X 0,Y 348.017,Z 335.13,A -85,B 0,C 180,E1 -14016.809,E2 -14016.809} C_VEL
LIN {X 0,Y 346.689,Z 349.525,A -85,B 0,C 180,E1 -14018.13,E2 -14018.13} C_VEL
LIN {X 0,Y 345.347,Z 362.887,A -85,B 0,C 180,E1 -14019.625,E2 -14019.625} C_VEL
LIN {X 0,Y 344.103,Z 374.865,A -85,B 0,C 180,E1 -14021.235,E2 -14021.235} C_VEL
LIN {X 0,Y 342.908,Z 386.015,A -85,B 0,C 180,E1 -14023.018,E2 -14023.018} C_VEL
LIN {X 0,Y 341.817,Z 396.101,A -85,B 0,C 180,E1 -14024.94,E2 -14024.94} C_VEL
LIN {X 0,Y 341.131,Z 404.704,A -85,B 0,C 180,E1 -14026.901,E2 -14026.901} C_VEL
LIN {X 0,Y 340.386,Z 411.377,A -85,B 0,C 180,E1 -14028.688,E2 -14028.688} C_VEL
LIN {X 0,Y 339.879,Z 418.645,A -85,B 0,C 180,E1 -14031.078,E2 -14031.078} C_VEL
LIN {X 0,Y 339.537,Z 424.358,A -85,B 0,C 180,E1 -14033.485,E2 -14033.485} C_VEL
LIN {X 0,Y 339.392,Z 427.598,A -85,B 0,C 180,E1 -14035.248,E2 -14035.248} C_VEL
LIN {X 0,Y 339.319,Z 430.8,A -85,B 0,C 180,E1 -14037.626,E2 -14037.626} C_VEL
LIN {X 0,Y 339.317,Z 432.714,A -85,B 0,C 180,E1 -14040,E2 -14040} C_VEL
